LIN {X 0,Y 573.208,Z 412.078,A -85,B 0,C 180,E1 -2311.434,E2 -2311.434} C_VEL
LIN {X 0,Y 573.228,Z 412.081,A -85,B 0,C 180,E1 -2314.589,E2 -2314.589} C_VEL
LIN {X 0,Y 573.218,Z 412.079,A -85,B 0,C 180,E1 -2317.661,E2 -2317.661} C_VEL
LIN {X 0,Y 573.204,Z 412.085,A -85,B 0,C 180,E1 -2319.921,E2 -2319.921} C_VEL
LIN {X 0,Y 573.193,Z 412.081,A -85,B 0,C 180,E1 -2323.014,E2 -2323.014} C_VEL
LIN {X 0,Y 573.247,Z 412.08,A -85,B 0,C 180,E1 -2325.806,E2 -2325.806} C_VEL
LIN {X 0,Y 573.224,Z 412.077,A -85,B 0,C 180,E1 -2328.768,E2 -2328.768} C_VEL
LIN {X 0,Y 573.234,Z 412.08,A -85,B 0,C 180,E1 -2331.54,E2 -2331.54} C_VEL
LIN {X 0,Y 573.262,Z 412.075,A -85,B 0,C 180,E1 -2334.371,E2 -2334.371} C_VEL
LIN {X 0,Y 573.309,Z 412.075,A -85,B 0,C 180,E1 -2337.892,E2 -2337.892} C_VEL
LIN {X 0,Y 573.268,Z 412.217,A -85,B 0,C 180,E1 -2339.122,E2 -2339.122} C_VEL
LIN {X 0,Y 573.209,Z 422.347,A -85,B 0,C 180,E1 -2341.229,E2 -2341.229} C_VEL
LIN {X 0,Y 574.074,Z 428.345,A -85,B 0,C 180,E1 -2341.337,E2 -2341.337} C_VEL
LIN {X 0,Y 573.848,Z 528.439,A -85,B 0,C 180,E1 -2342.61,E2 -2342.61} C_VEL
LIN {X 0,Y 573.75,Z 541.247,A -85,B 0,C 180,E1 -2342.918,E2 -2342.918} C_VEL
LIN {X 0,Y 573.682,Z 553.267,A -85,B 0,C 180,E1 -2343.336,E2 -2343.336} C_VEL
LIN {X 0,Y 573.54,Z 566.249,A -85,B 0,C 180,E1 -2343.952,E2 -2343.952} C_VEL
LIN {X 0,Y 573.376,Z 577.571,A -85,B 0,C 180,E1 -2344.658,E2 -2344.658} C_VEL
LIN {X 0,Y 573.327,Z 586.745,A -85,B 0,C 180,E1 -2345.363,E2 -2345.363} C_VEL
LIN {X 0,Y 573.226,Z 595.361,A -85,B 0,C 180,E1 -2346.158,E2 -2346.158} C_VEL
LIN {X 0,Y 573.165,Z 603.328,A -85,B 0,C 180,E1 -2347.043,E2 -2347.043} C_VEL
LIN {X 0,Y 573.122,Z 611.174,A -85,B 0,C 180,E1 -2348.107,E2 -2348.107} C_VEL
LIN {X 0,Y 573.018,Z 617.448,A -85,B 0,C 180,E1 -2349.175,E2 -2349.175} C_VEL
LIN {X 0,Y 573.002,Z 622.437,A -85,B 0,C 180,E1 -2350.244,E2 -2350.244} C_VEL
LIN {X 0,Y 572.984,Z 626.292,A -85,B 0,C 180,E1 -2351.318,E2 -2351.318} C_VEL
LIN {X 0,Y 572.952,Z 628.329,A -85,B 0,C 180,E1 -2352.036,E2 -2352.036} C_VEL
LIN {X 0,Y 572.946,Z 629.872,A -85,B 0,C 180,E1 -2352.756,E2 -2352.756} C_VEL
LIN {X 0,Y 572.981,Z 631.694,A -85,B 0,C 180,E1 -2354.2,E2 -2354.2} C_VEL
LIN {X 0,Y 572.906,Z 631.98,A -85,B 0,C 180,E1 -2354.928,E2 -2354.928} C_VEL
LIN {X 0,Y 572.917,Z 631.812,A -85,B 0,C 180,E1 -2355.657,E2 -2355.657} C_VEL
LIN {X 0,Y 572.942,Z 630.599,A -85,B 0,C 180,E1 -2356.904,E2 -2356.904} C_VEL
LIN {X 0,Y 572.952,Z 628.779,A -85,B 0,C 180,E1 -2357.858,E2 -2357.858} C_VEL
LIN {X 0,Y 572.974,Z 624.979,A -85,B 0,C 180,E1 -2359.183,E2 -2359.183} C_VEL
LIN {X 0,Y 573.014,Z 619.717,A -85,B 0,C 180,E1 -2360.46,E2 -2360.46} C_VEL
LIN {X 0,Y 573.092,Z 613.633,A -85,B 0,C 180,E1 -2361.586,E2 -2361.586} C_VEL
LIN {X 0,Y 573.121,Z 605.915,A -85,B 0,C 180,E1 -2362.723,E2 -2362.723} C_VEL
LIN {X 0,Y 573.121,Z 605.356,A -85,B 0,C 180,E1 -2362.795,E2 -2362.795} C_VEL
LIN {X 0,Y 572.463,Z 601.704,A -85,B 0,C 180,E1 -2363.256,E2 -2363.256} C_VEL
LIN {X 0,Y 569.645,Z 595.469,A -85,B 0,C 180,E1 -2363.977,E2 -2363.977} C_VEL
LIN {X 0,Y 566.893,Z 588.846,A -85,B 0,C 180,E1 -2364.659,E2 -2364.659} C_VEL
LIN {X 0,Y 566.352,Z 584.328,A -85,B 0,C 180,E1 -2365.053,E2 -2365.053} C_VEL
LIN {X 0,Y 566.483,Z 572.018,A -85,B 0,C 180,E1 -2365.933,E2 -2365.933} C_VEL
LIN {X 0,Y 566.64,Z 561.548,A -85,B 0,C 180,E1 -2366.52,E2 -2366.52} C_VEL
LIN {X 0,Y 566.736,Z 550.579,A -85,B 0,C 180,E1 -2367.005,E2 -2367.005} C_VEL
LIN {X 0,Y 566.849,Z 538.8,A -85,B 0,C 180,E1 -2367.393,E2 -2367.393} C_VEL
LIN {X 0,Y 566.936,Z 525.781,A -85,B 0,C 180,E1 -2367.677,E2 -2367.677} C_VEL
LIN {X 0,Y 567.085,Z 427.613,A -85,B 0,C 180,E1 -2368.934,E2 -2368.934} C_VEL
LIN {X 0,Y 566.174,Z 422.329,A -85,B 0,C 180,E1 -2369.039,E2 -2369.039} C_VEL
LIN {X 0,Y 566.194,Z 412.956,A -85,B 0,C 180,E1 -2371.048,E2 -2371.048} C_VEL
LIN {X 0,Y 566.2,Z 412.953,A -85,B 0,C 180,E1 -2373.732,E2 -2373.732} C_VEL
LIN {X 0,Y 566.177,Z 412.961,A -85,B 0,C 180,E1 -2376.572,E2 -2376.572} C_VEL
LIN {X 0,Y 566.212,Z 412.95,A -85,B 0,C 180,E1 -2379.685,E2 -2379.685} C_VEL
LIN {X 0,Y 566.195,Z 412.954,A -85,B 0,C 180,E1 -2382.916,E2 -2382.916} C_VEL
LIN {X 0,Y 566.159,Z 412.96,A -85,B 0,C 180,E1 -2386.053,E2 -2386.053} C_VEL
LIN {X 0,Y 566.16,Z 412.959,A -85,B 0,C 180,E1 -2388.859,E2 -2388.859} C_VEL
LIN {X 0,Y 566.204,Z 412.95,A -85,B 0,C 180,E1 -2391.443,E2 -2391.443} C_VEL
LIN {X 0,Y 566.145,Z 412.966,A -85,B 0,C 180,E1 -2394.306,E2 -2394.306} C_VEL
LIN {X 0,Y 566.213,Z 412.952,A -85,B 0,C 180,E1 -2396.897,E2 -2396.897} C_VEL
LIN {X 0,Y 566.171,Z 412.954,A -85,B 0,C 180,E1 -2399.406,E2 -2399.406} C_VEL
LIN {X 0,Y 566.172,Z 412.956,A -85,B 0,C 180,E1 -2401.855,E2 -2401.855} C_VEL
LIN {X 0,Y 566.196,Z 412.958,A -85,B 0,C 180,E1 -2404.25,E2 -2404.25} C_VEL
LIN {X 0,Y 566.168,Z 412.96,A -85,B 0,C 180,E1 -2406.72,E2 -2406.72} C_VEL
LIN {X 0,Y 566.204,Z 412.951,A -85,B 0,C 180,E1 -2409.662,E2 -2409.662} C_VEL
LIN {X 0,Y 566.178,Z 412.956,A -85,B 0,C 180,E1 -2411.921,E2 -2411.921} C_VEL
LIN {X 0,Y 566.189,Z 412.955,A -85,B 0,C 180,E1 -2414.89,E2 -2414.89} C_VEL
LIN {X 0,Y 566.214,Z 412.95,A -85,B 0,C 180,E1 -2417.818,E2 -2417.818} C_VEL
LIN {X 0,Y 566.174,Z 412.957,A -85,B 0,C 180,E1 -2419.992,E2 -2419.992} C_VEL
LIN {X 0,Y 566.213,Z 412.953,A -85,B 0,C 180,E1 -2422.87,E2 -2422.87} C_VEL
LIN {X 0,Y 566.263,Z 412.945,A -85,B 0,C 180,E1 -2425.016,E2 -2425.016} C_VEL
LIN {X 0,Y 566.281,Z 412.942,A -85,B 0,C 180,E1 -2427.866,E2 -2427.866} C_VEL
LIN {X 0,Y 566.299,Z 412.945,A -85,B 0,C 180,E1 -2430.711,E2 -2430.711} C_VEL
LIN {X 0,Y 566.26,Z 412.948,A -85,B 0,C 180,E1 -2432.845,E2 -2432.845} C_VEL
LIN {X 0,Y 566.247,Z 412.945,A -85,B 0,C 180,E1 -2435.698,E2 -2435.698} C_VEL
LIN {X 0,Y 566.194,Z 412.953,A -85,B 0,C 180,E1 -2437.847,E2 -2437.847} C_VEL
LIN {X 0,Y 566.236,Z 412.953,A -85,B 0,C 180,E1 -2440.73,E2 -2440.73} C_VEL
LIN {X 0,Y 566.189,Z 412.956,A -85,B 0,C 180,E1 -2442.91,E2 -2442.91} C_VEL
LIN {X 0,Y 566.196,Z 412.953,A -85,B 0,C 180,E1 -2445.109,E2 -2445.109} C_VEL
LIN {X 0,Y 566.195,Z 412.952,A -85,B 0,C 180,E1 -2447.332,E2 -2447.332} C_VEL
LIN {X 0,Y 566.207,Z 412.957,A -85,B 0,C 180,E1 -2450.337,E2 -2450.337} C_VEL
LIN {X 0,Y 566.169,Z 412.955,A -85,B 0,C 180,E1 -2453.28,E2 -2453.28} C_VEL
LIN {X 0,Y 566.204,Z 412.95,A -85,B 0,C 180,E1 -2455.749,E2 -2455.749} C_VEL
LIN {X 0,Y 566.184,Z 412.956,A -85,B 0,C 180,E1 -2458.954,E2 -2458.954} C_VEL
LIN {X 0,Y 566.192,Z 412.952,A -85,B 0,C 180,E1 -2461.422,E2 -2461.422} C_VEL
LIN {X 0,Y 566.208,Z 412.951,A -85,B 0,C 180,E1 -2463.956,E2 -2463.956} C_VEL
LIN {X 0,Y 566.182,Z 412.963,A -85,B 0,C 180,E1 -2466.571,E2 -2466.571} C_VEL
LIN {X 0,Y 566.211,Z 412.95,A -85,B 0,C 180,E1 -2469.274,E2 -2469.274} C_VEL
LIN {X 0,Y 566.187,Z 412.955,A -85,B 0,C 180,E1 -2472.09,E2 -2472.09} C_VEL
LIN {X 0,Y 566.167,Z 412.958,A -85,B 0,C 180,E1 -2475.036,E2 -2475.036} C_VEL
LIN {X 0,Y 566.186,Z 412.954,A -85,B 0,C 180,E1 -2477.91,E2 -2477.91} C_VEL
LIN {X 0,Y 566.211,Z 412.957,A -85,B 0,C 180,E1 -2480.726,E2 -2480.726} C_VEL
LIN {X 0,Y 566.181,Z 412.953,A -85,B 0,C 180,E1 -2483.429,E2 -2483.429} C_VEL
LIN {X 0,Y 566.211,Z 412.954,A -85,B 0,C 180,E1 -2486.266,E2 -2486.266} C_VEL
LIN {X 0,Y 566.189,Z 412.957,A -85,B 0,C 180,E1 -2488.924,E2 -2488.924} C_VEL
LIN {X 0,Y 566.191,Z 412.952,A -85,B 0,C 180,E1 -2491.856,E2 -2491.856} C_VEL
LIN {X 0,Y 566.237,Z 412.949,A -85,B 0,C 180,E1 -2495.039,E2 -2495.039} C_VEL
LIN {X 0,Y 566.191,Z 412.955,A -85,B 0,C 180,E1 -2498.137,E2 -2498.137} C_VEL
LIN {X 0,Y 566.23,Z 412.957,A -85,B 0,C 180,E1 -2500.614,E2 -2500.614} C_VEL
LIN {X 0,Y 566.207,Z 412.95,A -85,B 0,C 180,E1 -2503.412,E2 -2503.412} C_VEL
LIN {X 0,Y 566.19,Z 412.958,A -85,B 0,C 180,E1 -2506.359,E2 -2506.359} C_VEL
LIN {X 0,Y 566.235,Z 412.956,A -85,B 0,C 180,E1 -2508.675,E2 -2508.675} C_VEL
LIN {X 0,Y 566.225,Z 412.948,A -85,B 0,C 180,E1 -2511.434,E2 -2511.434} C_VEL
LIN {X 0,Y 566.262,Z 412.947,A -85,B 0,C 180,E1 -2514.302,E2 -2514.302} C_VEL
LIN {X 0,Y 566.282,Z 412.941,A -85,B 0,C 180,E1 -2517.866,E2 -2517.866} C_VEL
LIN {X 0,Y 566.303,Z 412.947,A -85,B 0,C 180,E1 -2520.711,E2 -2520.711} C_VEL
LIN {X 0,Y 566.27,Z 412.949,A -85,B 0,C 180,E1 -2522.846,E2 -2522.846} C_VEL
LIN {X 0,Y 566.251,Z 412.944,A -85,B 0,C 180,E1 -2525.698,E2 -2525.698} C_VEL
LIN {X 0,Y 566.227,Z 412.956,A -85,B 0,C 180,E1 -2528.566,E2 -2528.566} C_VEL
LIN {X 0,Y 566.242,Z 412.946,A -85,B 0,C 180,E1 -2531.454,E2 -2531.454} C_VEL
LIN {X 0,Y 566.235,Z 412.954,A -85,B 0,C 180,E1 -2534.507,E2 -2534.507} C_VEL
LIN {X 0,Y 566.199,Z 412.952,A -85,B 0,C 180,E1 -2537.332,E2 -2537.332} C_VEL
LIN {X 0,Y 566.208,Z 412.954,A -85,B 0,C 180,E1 -2540.337,E2 -2540.337} C_VEL
LIN {X 0,Y 566.17,Z 412.956,A -85,B 0,C 180,E1 -2543.281,E2 -2543.281} C_VEL
LIN {X 0,Y 566.206,Z 412.95,A -85,B 0,C 180,E1 -2545.749,E2 -2545.749} C_VEL
LIN {X 0,Y 566.188,Z 412.958,A -85,B 0,C 180,E1 -2548.954,E2 -2548.954} C_VEL
LIN {X 0,Y 566.193,Z 412.952,A -85,B 0,C 180,E1 -2551.422,E2 -2551.422} C_VEL
LIN {X 0,Y 566.209,Z 412.95,A -85,B 0,C 180,E1 -2553.956,E2 -2553.956} C_VEL
LIN {X 0,Y 566.201,Z 412.958,A -85,B 0,C 180,E1 -2556.57,E2 -2556.57} C_VEL
LIN {X 0,Y 566.214,Z 412.949,A -85,B 0,C 180,E1 -2559.686,E2 -2559.686} C_VEL
LIN {X 0,Y 566.202,Z 412.957,A -85,B 0,C 180,E1 -2562.917,E2 -2562.917} C_VEL
LIN {X 0,Y 566.199,Z 412.952,A -85,B 0,C 180,E1 -2566.049,E2 -2566.049} C_VEL
LIN {X 0,Y 566.205,Z 412.953,A -85,B 0,C 180,E1 -2569.215,E2 -2569.215} C_VEL
LIN {X 0,Y 566.187,Z 412.952,A -85,B 0,C 180,E1 -2571.637,E2 -2571.637} C_VEL
LIN {X 0,Y 566.151,Z 412.96,A -85,B 0,C 180,E1 -2574.307,E2 -2574.307} C_VEL
LIN {X 0,Y 566.221,Z 412.956,A -85,B 0,C 180,E1 -2576.898,E2 -2576.898} C_VEL
LIN {X 0,Y 566.181,Z 412.955,A -85,B 0,C 180,E1 -2579.407,E2 -2579.407} C_VEL
LIN {X 0,Y 566.214,Z 412.951,A -85,B 0,C 180,E1 -2581.858,E2 -2581.858} C_VEL
LIN {X 0,Y 566.221,Z 413.007,A -85,B 0,C 180,E1 -2584.733,E2 -2584.733} C_VEL
LIN {X 0,Y 567.446,Z 419.811,A -85,B 0,C 180,E1 -2585.682,E2 -2585.682} C_VEL
LIN {X 0,Y 567.201,Z 437.42,A -85,B 0,C 180,E1 -2587.987,E2 -2587.987} C_VEL
LIN {X 0,Y 566.912,Z 457.511,A -85,B 0,C 180,E1 -2590.633,E2 -2590.633} C_VEL
LIN {X 0,Y 566.69,Z 477.773,A -85,B 0,C 180,E1 -2593.264,E2 -2593.264} C_VEL
LIN {X 0,Y 566.458,Z 499.265,A -85,B 0,C 180,E1 -2595.988,E2 -2595.988} C_VEL
LIN {X 0,Y 567.166,Z 505.526,A -85,B 0,C 180,E1 -2596.086,E2 -2596.086} C_VEL
LIN {X 0,Y 566.957,Z 607.958,A -85,B 0,C 180,E1 -2597.403,E2 -2597.403} C_VEL
LIN {X 0,Y 566.847,Z 621.226,A -85,B 0,C 180,E1 -2597.719,E2 -2597.719} C_VEL
LIN {X 0,Y 566.719,Z 633.381,A -85,B 0,C 180,E1 -2598.148,E2 -2598.148} C_VEL
LIN {X 0,Y 566.629,Z 645.068,A -85,B 0,C 180,E1 -2598.704,E2 -2598.704} C_VEL
LIN {X 0,Y 566.5,Z 655.912,A -85,B 0,C 180,E1 -2599.366,E2 -2599.366} C_VEL
LIN {X 0,Y 566.335,Z 666.543,A -85,B 0,C 180,E1 -2600.176,E2 -2600.176} C_VEL
LIN {X 0,Y 566.207,Z 676.115,A -85,B 0,C 180,E1 -2601.074,E2 -2601.074} C_VEL
LIN {X 0,Y 566.112,Z 683.962,A -85,B 0,C 180,E1 -2601.972,E2 -2601.972} C_VEL
LIN {X 0,Y 566.003,Z 691.623,A -85,B 0,C 180,E1 -2603.047,E2 -2603.047} C_VEL
LIN {X 0,Y 566.004,Z 698.681,A -85,B 0,C 180,E1 -2604.299,E2 -2604.299} C_VEL
LIN {X 0,Y 565.933,Z 703.373,A -85,B 0,C 180,E1 -2605.37,E2 -2605.37} C_VEL
LIN {X 0,Y 565.927,Z 706.958,A -85,B 0,C 180,E1 -2606.44,E2 -2606.44} C_VEL
LIN {X 0,Y 565.878,Z 708.809,A -85,B 0,C 180,E1 -2607.153,E2 -2607.153} C_VEL
LIN {X 0,Y 565.846,Z 711.186,A -85,B 0,C 180,E1 -2608.577,E2 -2608.577} C_VEL
LIN {X 0,Y 565.839,Z 712,A -85,B 0,C 180,E1 -2610,E2 -2610} C_VEL
LIN {X 0,Y 565.846,Z 711.186,A -85,B 0,C 180,E1 -2611.424,E2 -2611.424} C_VEL
LIN {X 0,Y 565.878,Z 708.809,A -85,B 0,C 180,E1 -2612.848,E2 -2612.848} C_VEL
LIN {X 0,Y 565.926,Z 705.895,A -85,B 0,C 180,E1 -2613.917,E2 -2613.917} C_VEL
LIN {X 0,Y 565.878,Z 701.948,A -85,B 0,C 180,E1 -2614.988,E2 -2614.988} C_VEL
LIN {X 0,Y 566.002,Z 696.865,A -85,B 0,C 180,E1 -2616.059,E2 -2616.059} C_VEL
LIN {X 0,Y 566.04,Z 690.466,A -85,B 0,C 180,E1 -2617.133,E2 -2617.133} C_VEL
LIN {X 0,Y 566.134,Z 682.476,A -85,B 0,C 180,E1 -2618.208,E2 -2618.208} C_VEL
LIN {X 0,Y 566.229,Z 674.333,A -85,B 0,C 180,E1 -2619.106,E2 -2619.106} C_VEL
LIN {X 0,Y 566.345,Z 664.397,A -85,B 0,C 180,E1 -2620.005,E2 -2620.005} C_VEL
LIN {X 0,Y 566.53,Z 653.298,A -85,B 0,C 180,E1 -2620.807,E2 -2620.807} C_VEL
LIN {X 0,Y 566.613,Z 642.17,A -85,B 0,C 180,E1 -2621.447,E2 -2621.447} C_VEL
LIN {X 0,Y 566.722,Z 629.976,A -85,B 0,C 180,E1 -2621.989,E2 -2621.989} C_VEL
LIN {X 0,Y 566.882,Z 617.164,A -85,B 0,C 180,E1 -2622.394,E2 -2622.394} C_VEL
LIN {X 0,Y 566.963,Z 603.581,A -85,B 0,C 180,E1 -2622.665,E2 -2622.665} C_VEL
LIN {X 0,Y 567.027,Z 503.249,A -85,B 0,C 180,E1 -2623.947,E2 -2623.947} C_VEL
LIN {X 0,Y 566.442,Z 498.943,A -85,B 0,C 180,E1 -2624.024,E2 -2624.024} C_VEL
LIN {X 0,Y 566.708,Z 476.505,A -85,B 0,C 180,E1 -2626.9,E2 -2626.9} C_VEL
LIN {X 0,Y 566.959,Z 454.781,A -85,B 0,C 180,E1 -2629.724,E2 -2629.724} C_VEL
LIN {X 0,Y 567.29,Z 434.546,A -85,B 0,C 180,E1 -2632.393,E2 -2632.393} C_VEL
LIN {X 0,Y 567.403,Z 419.645,A -85,B 0,C 180,E1 -2634.321,E2 -2634.321} C_VEL
LIN {X 0,Y 566.219,Z 412.959,A -85,B 0,C 180,E1 -2635.263,E2 -2635.263} C_VEL
LIN {X 0,Y 566.207,Z 412.953,A -85,B 0,C 180,E1 -2638.202,E2 -2638.202} C_VEL
LIN {X 0,Y 566.195,Z 412.963,A -85,B 0,C 180,E1 -2641.076,E2 -2641.076} C_VEL
LIN {X 0,Y 566.216,Z 412.952,A -85,B 0,C 180,E1 -2643.734,E2 -2643.734} C_VEL
LIN {X 0,Y 566.203,Z 412.956,A -85,B 0,C 180,E1 -2646.57,E2 -2646.57} C_VEL
LIN {X 0,Y 566.219,Z 412.95,A -85,B 0,C 180,E1 -2649.686,E2 -2649.686} C_VEL
LIN {X 0,Y 566.202,Z 412.959,A -85,B 0,C 180,E1 -2652.917,E2 -2652.917} C_VEL
LIN {X 0,Y 566.198,Z 412.953,A -85,B 0,C 180,E1 -2656.049,E2 -2656.049} C_VEL
LIN {X 0,Y 566.207,Z 412.952,A -85,B 0,C 180,E1 -2659.215,E2 -2659.215} C_VEL
LIN {X 0,Y 566.184,Z 412.953,A -85,B 0,C 180,E1 -2661.637,E2 -2661.637} C_VEL
LIN {X 0,Y 566.147,Z 412.964,A -85,B 0,C 180,E1 -2664.307,E2 -2664.307} C_VEL
LIN {X 0,Y 566.215,Z 412.952,A -85,B 0,C 180,E1 -2666.897,E2 -2666.897} C_VEL
LIN {X 0,Y 566.172,Z 412.955,A -85,B 0,C 180,E1 -2669.407,E2 -2669.407} C_VEL
LIN {X 0,Y 566.174,Z 412.957,A -85,B 0,C 180,E1 -2671.855,E2 -2671.855} C_VEL
LIN {X 0,Y 566.19,Z 412.961,A -85,B 0,C 180,E1 -2674.25,E2 -2674.25} C_VEL
LIN {X 0,Y 566.163,Z 412.956,A -85,B 0,C 180,E1 -2677.368,E2 -2677.368} C_VEL
LIN {X 0,Y 566.154,Z 412.96,A -85,B 0,C 180,E1 -2679.661,E2 -2679.661} C_VEL
LIN {X 0,Y 566.152,Z 412.96,A -85,B 0,C 180,E1 -2682.667,E2 -2682.667} C_VEL
LIN {X 0,Y 566.217,Z 412.953,A -85,B 0,C 180,E1 -2685.626,E2 -2685.626} C_VEL
LIN {X 0,Y 566.19,Z 412.954,A -85,B 0,C 180,E1 -2688.701,E2 -2688.701} C_VEL
LIN {X 0,Y 566.185,Z 412.957,A -85,B 0,C 180,E1 -2691.434,E2 -2691.434} C_VEL
LIN {X 0,Y 566.232,Z 412.952,A -85,B 0,C 180,E1 -2694.301,E2 -2694.301} C_VEL
LIN {X 0,Y 566.28,Z 412.951,A -85,B 0,C 180,E1 -2697.866,E2 -2697.866} C_VEL
LIN {X 0,Y 566.225,Z 413.125,A -85,B 0,C 180,E1 -2699.111,E2 -2699.111} C_VEL
LIN {X 0,Y 566.196,Z 422.422,A -85,B 0,C 180,E1 -2701.067,E2 -2701.067} C_VEL
LIN {X 0,Y 567.178,Z 429.028,A -85,B 0,C 180,E1 -2701.176,E2 -2701.176} C_VEL
LIN {X 0,Y 566.932,Z 528.869,A -85,B 0,C 180,E1 -2702.464,E2 -2702.464} C_VEL
LIN {X 0,Y 566.791,Z 540.783,A -85,B 0,C 180,E1 -2702.754,E2 -2702.754} C_VEL
LIN {X 0,Y 566.745,Z 552.336,A -85,B 0,C 180,E1 -2703.154,E2 -2703.154} C_VEL
LIN {X 0,Y 566.614,Z 564.791,A -85,B 0,C 180,E1 -2703.734,E2 -2703.734} C_VEL
LIN {X 0,Y 566.42,Z 576.43,A -85,B 0,C 180,E1 -2704.448,E2 -2704.448} C_VEL
LIN {X 0,Y 566.342,Z 585.79,A -85,B 0,C 180,E1 -2705.162,E2 -2705.162} C_VEL
LIN {X 0,Y 566.181,Z 593.677,A -85,B 0,C 180,E1 -2705.878,E2 -2705.878} C_VEL
LIN {X 0,Y 566.14,Z 601.506,A -85,B 0,C 180,E1 -2706.726,E2 -2706.726} C_VEL
LIN {X 0,Y 566.06,Z 608.764,A -85,B 0,C 180,E1 -2707.67,E2 -2707.67} C_VEL
LIN {X 0,Y 565.977,Z 615.551,A -85,B 0,C 180,E1 -2708.749,E2 -2708.749} C_VEL
LIN {X 0,Y 565.94,Z 621.749,A -85,B 0,C 180,E1 -2710.012,E2 -2710.012} C_VEL
LIN {X 0,Y 565.914,Z 625.953,A -85,B 0,C 180,E1 -2711.159,E2 -2711.159} C_VEL
LIN {X 0,Y 565.869,Z 628.757,A -85,B 0,C 180,E1 -2712.189,E2 -2712.189} C_VEL
LIN {X 0,Y 565.845,Z 630.225,A -85,B 0,C 180,E1 -2712.919,E2 -2712.919} C_VEL
LIN {X 0,Y 565.854,Z 631.775,A -85,B 0,C 180,E1 -2714.355,E2 -2714.355} C_VEL
LIN {X 0,Y 565.808,Z 631.99,A -85,B 0,C 180,E1 -2715.12,E2 -2715.12} C_VEL
LIN {X 0,Y 565.812,Z 631.721,A -85,B 0,C 180,E1 -2715.859,E2 -2715.859} C_VEL
LIN {X 0,Y 565.858,Z 630.503,A -85,B 0,C 180,E1 -2716.991,E2 -2716.991} C_VEL
LIN {X 0,Y 565.893,Z 627.34,A -85,B 0,C 180,E1 -2718.463,E2 -2718.463} C_VEL
LIN {X 0,Y 565.889,Z 623.655,A -85,B 0,C 180,E1 -2719.592,E2 -2719.592} C_VEL
LIN {X 0,Y 565.948,Z 618.739,A -85,B 0,C 180,E1 -2720.727,E2 -2720.727} C_VEL
LIN {X 0,Y 566.009,Z 612.427,A -85,B 0,C 180,E1 -2721.87,E2 -2721.87} C_VEL
LIN {X 0,Y 566.074,Z 604.569,A -85,B 0,C 180,E1 -2722.996,E2 -2722.996} C_VEL
LIN {X 0,Y 566.185,Z 595.911,A -85,B 0,C 180,E1 -2723.987,E2 -2723.987} C_VEL
LIN {X 0,Y 566.28,Z 587.734,A -85,B 0,C 180,E1 -2724.763,E2 -2724.763} C_VEL
LIN {X 0,Y 566.352,Z 584.328,A -85,B 0,C 180,E1 -2725.053,E2 -2725.053} C_VEL
LIN {X 0,Y 565.807,Z 579.764,A -85,B 0,C 180,E1 -2725.428,E2 -2725.428} C_VEL
LIN {X 0,Y 563.079,Z 572.097,A -85,B 0,C 180,E1 -2726.003,E2 -2726.003} C_VEL
LIN {X 0,Y 560.399,Z 564.021,A -85,B 0,C 180,E1 -2726.524,E2 -2726.524} C_VEL
LIN {X 0,Y 559.712,Z 558.815,A -85,B 0,C 180,E1 -2726.799,E2 -2726.799} C_VEL
LIN {X 0,Y 559.838,Z 546.217,A -85,B 0,C 180,E1 -2727.322,E2 -2727.322} C_VEL
LIN {X 0,Y 559.97,Z 533.035,A -85,B 0,C 180,E1 -2727.695,E2 -2727.695} C_VEL
LIN {X 0,Y 560.063,Z 518.03,A -85,B 0,C 180,E1 -2727.944,E2 -2727.944} C_VEL
LIN {X 0,Y 560.181,Z 428.464,A -85,B 0,C 180,E1 -2729.098,E2 -2729.098} C_VEL
LIN {X 0,Y 559.125,Z 422.3,A -85,B 0,C 180,E1 -2729.226,E2 -2729.226} C_VEL
LIN {X 0,Y 559.16,Z 413.833,A -85,B 0,C 180,E1 -2731.051,E2 -2731.051} C_VEL
LIN {X 0,Y 559.158,Z 413.832,A -85,B 0,C 180,E1 -2733.947,E2 -2733.947} C_VEL
LIN {X 0,Y 559.127,Z 413.832,A -85,B 0,C 180,E1 -2737.11,E2 -2737.11} C_VEL
LIN {X 0,Y 559.16,Z 413.831,A -85,B 0,C 180,E1 -2739.941,E2 -2739.941} C_VEL
LIN {X 0,Y 559.152,Z 413.833,A -85,B 0,C 180,E1 -2742.744,E2 -2742.744} C_VEL
LIN {X 0,Y 559.126,Z 413.833,A -85,B 0,C 180,E1 -2745.764,E2 -2745.764} C_VEL
LIN {X 0,Y 559.123,Z 413.839,A -85,B 0,C 180,E1 -2748.226,E2 -2748.226} C_VEL
LIN {X 0,Y 559.172,Z 413.827,A -85,B 0,C 180,E1 -2751.192,E2 -2751.192} C_VEL
LIN {X 0,Y 559.118,Z 413.834,A -85,B 0,C 180,E1 -2753.787,E2 -2753.787} C_VEL
LIN {X 0,Y 559.163,Z 413.838,A -85,B 0,C 180,E1 -2756.425,E2 -2756.425} C_VEL
LIN {X 0,Y 559.151,Z 413.831,A -85,B 0,C 180,E1 -2758.98,E2 -2758.98} C_VEL
LIN {X 0,Y 559.119,Z 413.833,A -85,B 0,C 180,E1 -2761.629,E2 -2761.629} C_VEL
LIN {X 0,Y 559.16,Z 413.83,A -85,B 0,C 180,E1 -2763.902,E2 -2763.902} C_VEL
LIN {X 0,Y 559.137,Z 413.839,A -85,B 0,C 180,E1 -2766.573,E2 -2766.573} C_VEL
LIN {X 0,Y 559.175,Z 413.826,A -85,B 0,C 180,E1 -2769.395,E2 -2769.395} C_VEL
LIN {X 0,Y 559.127,Z 413.832,A -85,B 0,C 180,E1 -2771.685,E2 -2771.685} C_VEL
LIN {X 0,Y 559.141,Z 413.833,A -85,B 0,C 180,E1 -2773.947,E2 -2773.947} C_VEL
LIN {X 0,Y 559.158,Z 413.833,A -85,B 0,C 180,E1 -2776.183,E2 -2776.183} C_VEL
LIN {X 0,Y 559.193,Z 413.825,A -85,B 0,C 180,E1 -2779.133,E2 -2779.133} C_VEL
LIN {X 0,Y 559.192,Z 413.827,A -85,B 0,C 180,E1 -2782.053,E2 -2782.053} C_VEL
LIN {X 0,Y 559.239,Z 413.821,A -85,B 0,C 180,E1 -2784.953,E2 -2784.953} C_VEL
LIN {X 0,Y 559.252,Z 413.817,A -85,B 0,C 180,E1 -2787.839,E2 -2787.839} C_VEL
LIN {X 0,Y 559.269,Z 413.82,A -85,B 0,C 180,E1 -2790.72,E2 -2790.72} C_VEL
LIN {X 0,Y 559.226,Z 413.823,A -85,B 0,C 180,E1 -2792.881,E2 -2792.881} C_VEL
LIN {X 0,Y 559.218,Z 413.821,A -85,B 0,C 180,E1 -2795.77,E2 -2795.77} C_VEL
LIN {X 0,Y 559.168,Z 413.834,A -85,B 0,C 180,E1 -2798.674,E2 -2798.674} C_VEL
LIN {X 0,Y 559.206,Z 413.822,A -85,B 0,C 180,E1 -2801.6,E2 -2801.6} C_VEL
LIN {X 0,Y 559.202,Z 413.831,A -85,B 0,C 180,E1 -2804.595,E2 -2804.595} C_VEL
LIN {X 0,Y 559.138,Z 413.83,A -85,B 0,C 180,E1 -2807.557,E2 -2807.557} C_VEL
LIN {X 0,Y 559.167,Z 413.828,A -85,B 0,C 180,E1 -2809.837,E2 -2809.837} C_VEL
LIN {X 0,Y 559.14,Z 413.834,A -85,B 0,C 180,E1 -2812.153,E2 -2812.153} C_VEL
LIN {X 0,Y 559.175,Z 413.826,A -85,B 0,C 180,E1 -2815.298,E2 -2815.298} C_VEL
LIN {X 0,Y 559.127,Z 413.832,A -85,B 0,C 180,E1 -2817.715,E2 -2817.715} C_VEL
LIN {X 0,Y 559.152,Z 413.833,A -85,B 0,C 180,E1 -2820.183,E2 -2820.183} C_VEL
LIN {X 0,Y 559.153,Z 413.836,A -85,B 0,C 180,E1 -2822.715,E2 -2822.715} C_VEL
LIN {X 0,Y 559.122,Z 413.833,A -85,B 0,C 180,E1 -2825.324,E2 -2825.324} C_VEL
LIN {X 0,Y 559.13,Z 413.833,A -85,B 0,C 180,E1 -2828.018,E2 -2828.018} C_VEL
LIN {X 0,Y 559.155,Z 413.834,A -85,B 0,C 180,E1 -2830.812,E2 -2830.812} C_VEL
LIN {X 0,Y 559.111,Z 413.834,A -85,B 0,C 180,E1 -2833.737,E2 -2833.737} C_VEL
LIN {X 0,Y 559.136,Z 413.836,A -85,B 0,C 180,E1 -2836.266,E2 -2836.266} C_VEL
LIN {X 0,Y 559.155,Z 413.83,A -85,B 0,C 180,E1 -2839.187,E2 -2839.187} C_VEL
LIN {X 0,Y 559.129,Z 413.833,A -85,B 0,C 180,E1 -2841.982,E2 -2841.982} C_VEL
LIN {X 0,Y 559.128,Z 413.838,A -85,B 0,C 180,E1 -2844.788,E2 -2844.788} C_VEL
LIN {X 0,Y 559.155,Z 413.829,A -85,B 0,C 180,E1 -2847.365,E2 -2847.365} C_VEL
LIN {X 0,Y 559.147,Z 413.832,A -85,B 0,C 180,E1 -2850.143,E2 -2850.143} C_VEL
LIN {X 0,Y 559.159,Z 413.83,A -85,B 0,C 180,E1 -2853.175,E2 -2853.175} C_VEL
LIN {X 0,Y 559.157,Z 413.828,A -85,B 0,C 180,E1 -2855.495,E2 -2855.495} C_VEL
LIN {X 0,Y 559.171,Z 413.837,A -85,B 0,C 180,E1 -2858.624,E2 -2858.624} C_VEL
LIN {X 0,Y 559.16,Z 413.833,A -85,B 0,C 180,E1 -2860.926,E2 -2860.926} C_VEL
LIN {X 0,Y 559.156,Z 413.829,A -85,B 0,C 180,E1 -2863.948,E2 -2863.948} C_VEL
LIN {X 0,Y 559.163,Z 413.83,A -85,B 0,C 180,E1 -2866.184,E2 -2866.184} C_VEL
LIN {X 0,Y 559.206,Z 413.832,A -85,B 0,C 180,E1 -2868.605,E2 -2868.605} C_VEL
LIN {X 0,Y 559.203,Z 413.824,A -85,B 0,C 180,E1 -2872.054,E2 -2872.054} C_VEL
LIN {X 0,Y 559.247,Z 413.822,A -85,B 0,C 180,E1 -2874.953,E2 -2874.953} C_VEL
LIN {X 0,Y 559.253,Z 413.816,A -85,B 0,C 180,E1 -2877.839,E2 -2877.839} C_VEL
LIN {X 0,Y 559.273,Z 413.823,A -85,B 0,C 180,E1 -2880.72,E2 -2880.72} C_VEL
LIN {X 0,Y 559.236,Z 413.824,A -85,B 0,C 180,E1 -2882.881,E2 -2882.881} C_VEL
LIN {X 0,Y 559.222,Z 413.82,A -85,B 0,C 180,E1 -2885.77,E2 -2885.77} C_VEL
LIN {X 0,Y 559.186,Z 413.835,A -85,B 0,C 180,E1 -2888.674,E2 -2888.674} C_VEL
LIN {X 0,Y 559.206,Z 413.822,A -85,B 0,C 180,E1 -2891.601,E2 -2891.601} C_VEL
LIN {X 0,Y 559.201,Z 413.831,A -85,B 0,C 180,E1 -2894.596,E2 -2894.596} C_VEL
LIN {X 0,Y 559.143,Z 413.83,A -85,B 0,C 180,E1 -2897.558,E2 -2897.558} C_VEL
LIN {X 0,Y 559.166,Z 413.827,A -85,B 0,C 180,E1 -2899.838,E2 -2899.838} C_VEL
LIN {X 0,Y 559.141,Z 413.832,A -85,B 0,C 180,E1 -2902.153,E2 -2902.153} C_VEL
LIN {X 0,Y 559.175,Z 413.827,A -85,B 0,C 180,E1 -2905.298,E2 -2905.298} C_VEL
LIN {X 0,Y 559.168,Z 413.831,A -85,B 0,C 180,E1 -2908.381,E2 -2908.381} C_VEL
LIN {X 0,Y 559.146,Z 413.831,A -85,B 0,C 180,E1 -2911.273,E2 -2911.273} C_VEL
LIN {X 0,Y 559.166,Z 413.827,A -85,B 0,C 180,E1 -2913.949,E2 -2913.949} C_VEL
LIN {X 0,Y 559.141,Z 413.834,A -85,B 0,C 180,E1 -2917.109,E2 -2917.109} C_VEL
LIN {X 0,Y 559.16,Z 413.828,A -85,B 0,C 180,E1 -2919.942,E2 -2919.942} C_VEL
LIN {X 0,Y 559.158,Z 413.838,A -85,B 0,C 180,E1 -2922.744,E2 -2922.744} C_VEL
LIN {X 0,Y 559.152,Z 413.829,A -85,B 0,C 180,E1 -2925.761,E2 -2925.761} C_VEL
LIN {X 0,Y 559.164,Z 413.83,A -85,B 0,C 180,E1 -2928.23,E2 -2928.23} C_VEL
LIN {X 0,Y 559.177,Z 413.829,A -85,B 0,C 180,E1 -2931.192,E2 -2931.192} C_VEL
LIN {X 0,Y 559.123,Z 413.832,A -85,B 0,C 180,E1 -2933.788,E2 -2933.788} C_VEL
LIN {X 0,Y 559.164,Z 413.832,A -85,B 0,C 180,E1 -2936.425,E2 -2936.425} C_VEL
LIN {X 0,Y 559.156,Z 413.835,A -85,B 0,C 180,E1 -2938.981,E2 -2938.981} C_VEL
LIN {X 0,Y 559.147,Z 413.832,A -85,B 0,C 180,E1 -2941.623,E2 -2941.623} C_VEL
LIN {X 0,Y 559.212,Z 413.994,A -85,B 0,C 180,E1 -2944.579,E2 -2944.579} C_VEL
LIN {X 0,Y 560.507,Z 420.864,A -85,B 0,C 180,E1 -2945.558,E2 -2945.558} C_VEL
LIN {X 0,Y 560.272,Z 438.578,A -85,B 0,C 180,E1 -2947.894,E2 -2947.894} C_VEL
LIN {X 0,Y 559.98,Z 459.286,A -85,B 0,C 180,E1 -2950.62,E2 -2950.62} C_VEL
LIN {X 0,Y 559.68,Z 481.906,A -85,B 0,C 180,E1 -2953.589,E2 -2953.589} C_VEL
LIN {X 0,Y 559.501,Z 499.265,A -85,B 0,C 180,E1 -2955.81,E2 -2955.81} C_VEL
LIN {X 0,Y 560.278,Z 506.196,A -85,B 0,C 180,E1 -2955.92,E2 -2955.92} C_VEL
LIN {X 0,Y 560.027,Z 607.958,A -85,B 0,C 180,E1 -2957.245,E2 -2957.245} C_VEL
LIN {X 0,Y 559.904,Z 621.226,A -85,B 0,C 180,E1 -2957.564,E2 -2957.564} C_VEL
LIN {X 0,Y 559.766,Z 633.382,A -85,B 0,C 180,E1 -2957.999,E2 -2957.999} C_VEL
LIN {X 0,Y 559.668,Z 644.813,A -85,B 0,C 180,E1 -2958.547,E2 -2958.547} C_VEL
LIN {X 0,Y 559.516,Z 655.91,A -85,B 0,C 180,E1 -2959.232,E2 -2959.232} C_VEL
LIN {X 0,Y 559.315,Z 666.542,A -85,B 0,C 180,E1 -2960.051,E2 -2960.051} C_VEL
LIN {X 0,Y 559.161,Z 676.115,A -85,B 0,C 180,E1 -2960.961,E2 -2960.961} C_VEL
LIN {X 0,Y 559.05,Z 683.962,A -85,B 0,C 180,E1 -2961.87,E2 -2961.87} C_VEL
LIN {X 0,Y 558.943,Z 691.624,A -85,B 0,C 180,E1 -2962.959,E2 -2962.959} C_VEL
LIN {X 0,Y 558.935,Z 698.681,A -85,B 0,C 180,E1 -2964.227,E2 -2964.227} C_VEL
LIN {X 0,Y 558.826,Z 703.373,A -85,B 0,C 180,E1 -2965.311,E2 -2965.311} C_VEL
LIN {X 0,Y 558.836,Z 706.958,A -85,B 0,C 180,E1 -2966.395,E2 -2966.395} C_VEL
LIN {X 0,Y 558.799,Z 708.808,A -85,B 0,C 180,E1 -2967.117,E2 -2967.117} C_VEL
LIN {X 0,Y 558.745,Z 711.185,A -85,B 0,C 180,E1 -2968.559,E2 -2968.559} C_VEL
LIN {X 0,Y 558.74,Z 712,A -85,B 0,C 180,E1 -2970,E2 -2970} C_VEL
LIN {X 0,Y 558.745,Z 711.185,A -85,B 0,C 180,E1 -2971.442,E2 -2971.442} C_VEL
LIN {X 0,Y 558.799,Z 708.809,A -85,B 0,C 180,E1 -2972.884,E2 -2972.884} C_VEL
LIN {X 0,Y 558.844,Z 705.895,A -85,B 0,C 180,E1 -2973.966,E2 -2973.966} C_VEL
LIN {X 0,Y 558.798,Z 701.948,A -85,B 0,C 180,E1 -2975.051,E2 -2975.051} C_VEL
LIN {X 0,Y 558.921,Z 696.865,A -85,B 0,C 180,E1 -2976.136,E2 -2976.136} C_VEL
LIN {X 0,Y 558.978,Z 690.466,A -85,B 0,C 180,E1 -2977.223,E2 -2977.223} C_VEL
LIN {X 0,Y 559.099,Z 682.475,A -85,B 0,C 180,E1 -2978.312,E2 -2978.312} C_VEL
LIN {X 0,Y 559.185,Z 674.332,A -85,B 0,C 180,E1 -2979.221,E2 -2979.221} C_VEL
LIN {X 0,Y 559.355,Z 664.396,A -85,B 0,C 180,E1 -2980.131,E2 -2980.131} C_VEL
LIN {X 0,Y 559.534,Z 653.4,A -85,B 0,C 180,E1 -2980.937,E2 -2980.937} C_VEL
LIN {X 0,Y 559.672,Z 641.455,A -85,B 0,C 180,E1 -2981.628,E2 -2981.628} C_VEL
LIN {X 0,Y 559.817,Z 628.759,A -85,B 0,C 180,E1 -2982.185,E2 -2982.185} C_VEL
LIN {X 0,Y 559.967,Z 615.334,A -85,B 0,C 180,E1 -2982.596,E2 -2982.596} C_VEL
LIN {X 0,Y 560.072,Z 602.062,A -85,B 0,C 180,E1 -2982.847,E2 -2982.847} C_VEL
LIN {X 0,Y 560.245,Z 504.935,A -85,B 0,C 180,E1 -2984.097,E2 -2984.097} C_VEL
LIN {X 0,Y 559.458,Z 498.943,A -85,B 0,C 180,E1 -2984.203,E2 -2984.203} C_VEL
LIN {X 0,Y 559.735,Z 476.827,A -85,B 0,C 180,E1 -2987.074,E2 -2987.074} C_VEL
LIN {X 0,Y 560.04,Z 456.072,A -85,B 0,C 180,E1 -2989.806,E2 -2989.806} C_VEL
LIN {X 0,Y 560.214,Z 440.013,A -85,B 0,C 180,E1 -2991.907,E2 -2991.907} C_VEL
LIN {X 0,Y 560.501,Z 422.028,A -85,B 0,C 180,E1 -2994.246,E2 -2994.246} C_VEL
LIN {X 0,Y 559.898,Z 417.471,A -85,B 0,C 180,E1 -2994.867,E2 -2994.867} C_VEL
LIN {X 0,Y 559.188,Z 413.834,A -85,B 0,C 180,E1 -2995.398,E2 -2995.398} C_VEL
LIN {X 0,Y 559.172,Z 413.83,A -85,B 0,C 180,E1 -2998.381,E2 -2998.381} C_VEL
LIN {X 0,Y 559.15,Z 413.838,A -85,B 0,C 180,E1 -3001.273,E2 -3001.273} C_VEL
LIN {X 0,Y 559.17,Z 413.829,A -85,B 0,C 180,E1 -3003.949,E2 -3003.949} C_VEL
LIN {X 0,Y 559.145,Z 413.837,A -85,B 0,C 180,E1 -3007.109,E2 -3007.109} C_VEL
LIN {X 0,Y 559.164,Z 413.829,A -85,B 0,C 180,E1 -3009.942,E2 -3009.942} C_VEL
LIN {X 0,Y 559.159,Z 413.838,A -85,B 0,C 180,E1 -3012.744,E2 -3012.744} C_VEL
LIN {X 0,Y 559.153,Z 413.829,A -85,B 0,C 180,E1 -3015.761,E2 -3015.761} C_VEL
LIN {X 0,Y 559.164,Z 413.831,A -85,B 0,C 180,E1 -3018.23,E2 -3018.23} C_VEL
LIN {X 0,Y 559.175,Z 413.828,A -85,B 0,C 180,E1 -3021.192,E2 -3021.192} C_VEL
LIN {X 0,Y 559.122,Z 413.833,A -85,B 0,C 180,E1 -3023.788,E2 -3023.788} C_VEL
LIN {X 0,Y 559.164,Z 413.836,A -85,B 0,C 180,E1 -3026.425,E2 -3026.425} C_VEL
LIN {X 0,Y 559.153,Z 413.831,A -85,B 0,C 180,E1 -3028.98,E2 -3028.98} C_VEL
LIN {X 0,Y 559.119,Z 413.834,A -85,B 0,C 180,E1 -3031.629,E2 -3031.629} C_VEL
LIN {X 0,Y 559.13,Z 413.836,A -85,B 0,C 180,E1 -3034.699,E2 -3034.699} C_VEL
LIN {X 0,Y 559.114,Z 413.835,A -85,B 0,C 180,E1 -3037.066,E2 -3037.066} C_VEL
LIN {X 0,Y 559.114,Z 413.835,A -85,B 0,C 180,E1 -3039.393,E2 -3039.393} C_VEL
LIN {X 0,Y 559.109,Z 413.84,A -85,B 0,C 180,E1 -3042.441,E2 -3042.441} C_VEL
LIN {X 0,Y 559.155,Z 413.831,A -85,B 0,C 180,E1 -3045.441,E2 -3045.441} C_VEL
LIN {X 0,Y 559.146,Z 413.832,A -85,B 0,C 180,E1 -3048.638,E2 -3048.638} C_VEL
LIN {X 0,Y 559.15,Z 413.832,A -85,B 0,C 180,E1 -3051.325,E2 -3051.325} C_VEL
LIN {X 0,Y 559.201,Z 413.829,A -85,B 0,C 180,E1 -3054.229,E2 -3054.229} C_VEL
LIN {X 0,Y 559.25,Z 413.827,A -85,B 0,C 180,E1 -3057.839,E2 -3057.839} C_VEL
LIN {X 0,Y 559.188,Z 413.928,A -85,B 0,C 180,E1 -3059.077,E2 -3059.077} C_VEL
LIN {X 0,Y 559.137,Z 422.362,A -85,B 0,C 180,E1 -3060.878,E2 -3060.878} C_VEL
LIN {X 0,Y 560.283,Z 429.716,A -85,B 0,C 180,E1 -3061.011,E2 -3061.011} C_VEL
LIN {X 0,Y 560.019,Z 528.118,A -85,B 0,C 180,E1 -3062.293,E2 -3062.293} C_VEL
LIN {X 0,Y 559.897,Z 540.264,A -85,B 0,C 180,E1 -3062.585,E2 -3062.585} C_VEL
LIN {X 0,Y 559.786,Z 550.266,A -85,B 0,C 180,E1 -3062.924,E2 -3062.924} C_VEL
LIN {X 0,Y 559.711,Z 559.577,A -85,B 0,C 180,E1 -3063.329,E2 -3063.329} C_VEL
LIN {X 0,Y 559.537,Z 569.557,A -85,B 0,C 180,E1 -3063.871,E2 -3063.871} C_VEL
LIN {X 0,Y 559.362,Z 579.041,A -85,B 0,C 180,E1 -3064.504,E2 -3064.504} C_VEL
LIN {X 0,Y 559.278,Z 587.989,A -85,B 0,C 180,E1 -3065.227,E2 -3065.227} C_VEL
LIN {X 0,Y 559.121,Z 597.303,A -85,B 0,C 180,E1 -3066.133,E2 -3066.133} C_VEL
LIN {X 0,Y 559.025,Z 606.278,A -85,B 0,C 180,E1 -3067.222,E2 -3067.222} C_VEL
LIN {X 0,Y 558.942,Z 613.477,A -85,B 0,C 180,E1 -3068.314,E2 -3068.314} C_VEL
LIN {X 0,Y 558.838,Z 619.301,A -85,B 0,C 180,E1 -3069.409,E2 -3069.409} C_VEL
LIN {X 0,Y 558.829,Z 623.903,A -85,B 0,C 180,E1 -3070.507,E2 -3070.507} C_VEL
LIN {X 0,Y 558.799,Z 627.41,A -85,B 0,C 180,E1 -3071.609,E2 -3071.609} C_VEL
LIN {X 0,Y 558.745,Z 630.521,A -85,B 0,C 180,E1 -3073.086,E2 -3073.086} C_VEL
LIN {X 0,Y 558.762,Z 631.798,A -85,B 0,C 180,E1 -3074.42,E2 -3074.42} C_VEL
LIN {X 0,Y 558.711,Z 631.942,A -85,B 0,C 180,E1 -3075.317,E2 -3075.317} C_VEL
LIN {X 0,Y 558.729,Z 631.596,A -85,B 0,C 180,E1 -3076.065,E2 -3076.065} C_VEL
LIN {X 0,Y 558.767,Z 630.41,A -85,B 0,C 180,E1 -3077.077,E2 -3077.077} C_VEL
LIN {X 0,Y 558.779,Z 627.847,A -85,B 0,C 180,E1 -3078.327,E2 -3078.327} C_VEL
LIN {X 0,Y 558.804,Z 624.628,A -85,B 0,C 180,E1 -3079.392,E2 -3079.392} C_VEL
LIN {X 0,Y 558.844,Z 619.604,A -85,B 0,C 180,E1 -3080.617,E2 -3080.617} C_VEL
LIN {X 0,Y 558.931,Z 615.149,A -85,B 0,C 180,E1 -3081.49,E2 -3081.49} C_VEL
LIN {X 0,Y 558.981,Z 608.51,A -85,B 0,C 180,E1 -3082.549,E2 -3082.549} C_VEL
LIN {X 0,Y 559.095,Z 601.026,A -85,B 0,C 180,E1 -3083.526,E2 -3083.526} C_VEL
LIN {X 0,Y 559.181,Z 593.88,A -85,B 0,C 180,E1 -3084.306,E2 -3084.306} C_VEL
LIN {X 0,Y 559.334,Z 584.742,A -85,B 0,C 180,E1 -3085.143,E2 -3085.143} C_VEL
LIN {X 0,Y 559.457,Z 573.418,A -85,B 0,C 180,E1 -3085.983,E2 -3085.983} C_VEL
LIN {X 0,Y 559.665,Z 562.33,A -85,B 0,C 180,E1 -3086.625,E2 -3086.625} C_VEL
LIN {X 0,Y 559.712,Z 558.815,A -85,B 0,C 180,E1 -3086.799,E2 -3086.799} C_VEL
LIN {X 0,Y 559.144,Z 553.503,A -85,B 0,C 180,E1 -3087.058,E2 -3087.058} C_VEL
LIN {X 0,Y 556.451,Z 544.755,A -85,B 0,C 180,E1 -3087.45,E2 -3087.45} C_VEL
LIN {X 0,Y 553.774,Z 535.764,A -85,B 0,C 180,E1 -3087.776,E2 -3087.776} C_VEL
LIN {X 0,Y 553.102,Z 530.074,A -85,B 0,C 180,E1 -3087.92,E2 -3087.92} C_VEL
LIN {X 0,Y 553.204,Z 505.728,A -85,B 0,C 180,E1 -3088.268,E2 -3088.268} C_VEL
LIN {X 0,Y 553.388,Z 429.806,A -85,B 0,C 180,E1 -3089.257,E2 -3089.257} C_VEL
LIN {X 0,Y 552.05,Z 422.345,A -85,B 0,C 180,E1 -3089.402,E2 -3089.402} C_VEL
LIN {X 0,Y 552.133,Z 414.708,A -85,B 0,C 180,E1 -3091.085,E2 -3091.085} C_VEL
LIN {X 0,Y 552.102,Z 414.715,A -85,B 0,C 180,E1 -3094.165,E2 -3094.165} C_VEL
LIN {X 0,Y 552.098,Z 414.712,A -85,B 0,C 180,E1 -3096.748,E2 -3096.748} C_VEL
LIN {X 0,Y 552.129,Z 414.704,A -85,B 0,C 180,E1 -3099.527,E2 -3099.527} C_VEL
LIN {X 0,Y 552.112,Z 414.716,A -85,B 0,C 180,E1 -3102.427,E2 -3102.427} C_VEL
LIN {X 0,Y 552.077,Z 414.71,A -85,B 0,C 180,E1 -3105.56,E2 -3105.56} C_VEL
LIN {X 0,Y 552.083,Z 414.715,A -85,B 0,C 180,E1 -3108.683,E2 -3108.683} C_VEL
LIN {X 0,Y 552.114,Z 414.705,A -85,B 0,C 180,E1 -3111.41,E2 -3111.41} C_VEL
LIN {X 0,Y 552.068,Z 414.719,A -85,B 0,C 180,E1 -3114.562,E2 -3114.562} C_VEL
LIN {X 0,Y 552.115,Z 414.706,A -85,B 0,C 180,E1 -3117.154,E2 -3117.154} C_VEL
LIN {X 0,Y 552.099,Z 414.71,A -85,B 0,C 180,E1 -3119.953,E2 -3119.953} C_VEL
LIN {X 0,Y 552.095,Z 414.71,A -85,B 0,C 180,E1 -3123.009,E2 -3123.009} C_VEL
LIN {X 0,Y 552.087,Z 414.711,A -85,B 0,C 180,E1 -3125.961,E2 -3125.961} C_VEL
LIN {X 0,Y 552.118,Z 414.706,A -85,B 0,C 180,E1 -3129.119,E2 -3129.119} C_VEL
LIN {X 0,Y 552.087,Z 414.709,A -85,B 0,C 180,E1 -3131.443,E2 -3131.443} C_VEL
LIN {X 0,Y 552.088,Z 414.709,A -85,B 0,C 180,E1 -3133.736,E2 -3133.736} C_VEL
LIN {X 0,Y 552.127,Z 414.707,A -85,B 0,C 180,E1 -3136.004,E2 -3136.004} C_VEL
LIN {X 0,Y 552.162,Z 414.702,A -85,B 0,C 180,E1 -3138.993,E2 -3138.993} C_VEL
LIN {X 0,Y 552.147,Z 414.704,A -85,B 0,C 180,E1 -3141.951,E2 -3141.951} C_VEL
LIN {X 0,Y 552.215,Z 414.696,A -85,B 0,C 180,E1 -3144.889,E2 -3144.889} C_VEL
LIN {X 0,Y 552.223,Z 414.693,A -85,B 0,C 180,E1 -3147.812,E2 -3147.812} C_VEL
LIN {X 0,Y 552.24,Z 414.696,A -85,B 0,C 180,E1 -3150.729,E2 -3150.729} C_VEL
LIN {X 0,Y 552.192,Z 414.699,A -85,B 0,C 180,E1 -3152.918,E2 -3152.918} C_VEL
LIN {X 0,Y 552.191,Z 414.697,A -85,B 0,C 180,E1 -3155.844,E2 -3155.844} C_VEL
LIN {X 0,Y 552.139,Z 414.708,A -85,B 0,C 180,E1 -3158.786,E2 -3158.786} C_VEL
LIN {X 0,Y 552.163,Z 414.7,A -85,B 0,C 180,E1 -3161.75,E2 -3161.75} C_VEL
LIN {X 0,Y 552.137,Z 414.709,A -85,B 0,C 180,E1 -3164.748,E2 -3164.748} C_VEL
LIN {X 0,Y 552.097,Z 414.708,A -85,B 0,C 180,E1 -3167.789,E2 -3167.789} C_VEL
LIN {X 0,Y 552.127,Z 414.707,A -85,B 0,C 180,E1 -3170.101,E2 -3170.101} C_VEL
LIN {X 0,Y 552.091,Z 414.717,A -85,B 0,C 180,E1 -3172.451,E2 -3172.451} C_VEL
LIN {X 0,Y 552.138,Z 414.703,A -85,B 0,C 180,E1 -3175.346,E2 -3175.346} C_VEL
LIN {X 0,Y 552.078,Z 414.713,A -85,B 0,C 180,E1 -3178.1,E2 -3178.1} C_VEL
LIN {X 0,Y 552.101,Z 414.716,A -85,B 0,C 180,E1 -3180.609,E2 -3180.609} C_VEL
LIN {X 0,Y 552.112,Z 414.707,A -85,B 0,C 180,E1 -3183.186,E2 -3183.186} C_VEL
LIN {X 0,Y 552.075,Z 414.711,A -85,B 0,C 180,E1 -3185.844,E2 -3185.844} C_VEL
LIN {X 0,Y 552.116,Z 414.715,A -85,B 0,C 180,E1 -3188.589,E2 -3188.589} C_VEL
LIN {X 0,Y 552.12,Z 414.705,A -85,B 0,C 180,E1 -3191.446,E2 -3191.446} C_VEL
LIN {X 0,Y 552.078,Z 414.72,A -85,B 0,C 180,E1 -3194.53,E2 -3194.53} C_VEL
LIN {X 0,Y 552.109,Z 414.706,A -85,B 0,C 180,E1 -3197.587,E2 -3197.587} C_VEL
LIN {X 0,Y 552.128,Z 414.712,A -85,B 0,C 180,E1 -3200.473,E2 -3200.473} C_VEL
LIN {X 0,Y 552.098,Z 414.708,A -85,B 0,C 180,E1 -3203.318,E2 -3203.318} C_VEL
LIN {X 0,Y 552.125,Z 414.705,A -85,B 0,C 180,E1 -3205.939,E2 -3205.939} C_VEL
LIN {X 0,Y 552.119,Z 414.714,A -85,B 0,C 180,E1 -3208.541,E2 -3208.541} C_VEL
LIN {X 0,Y 552.104,Z 414.707,A -85,B 0,C 180,E1 -3211.442,E2 -3211.442} C_VEL
LIN {X 0,Y 552.123,Z 414.71,A -85,B 0,C 180,E1 -3214.355,E2 -3214.355} C_VEL
LIN {X 0,Y 552.098,Z 414.715,A -85,B 0,C 180,E1 -3216.758,E2 -3216.758} C_VEL
LIN {X 0,Y 552.117,Z 414.708,A -85,B 0,C 180,E1 -3219.12,E2 -3219.12} C_VEL
LIN {X 0,Y 552.118,Z 414.705,A -85,B 0,C 180,E1 -3221.444,E2 -3221.444} C_VEL
LIN {X 0,Y 552.108,Z 414.706,A -85,B 0,C 180,E1 -3223.737,E2 -3223.737} C_VEL
LIN {X 0,Y 552.13,Z 414.705,A -85,B 0,C 180,E1 -3226.004,E2 -3226.004} C_VEL
LIN {X 0,Y 552.161,Z 414.704,A -85,B 0,C 180,E1 -3228.993,E2 -3228.993} C_VEL
LIN {X 0,Y 552.157,Z 414.701,A -85,B 0,C 180,E1 -3231.952,E2 -3231.952} C_VEL
LIN {X 0,Y 552.223,Z 414.698,A -85,B 0,C 180,E1 -3234.889,E2 -3234.889} C_VEL
LIN {X 0,Y 552.224,Z 414.692,A -85,B 0,C 180,E1 -3237.812,E2 -3237.812} C_VEL
LIN {X 0,Y 552.243,Z 414.698,A -85,B 0,C 180,E1 -3240.729,E2 -3240.729} C_VEL
LIN {X 0,Y 552.202,Z 414.7,A -85,B 0,C 180,E1 -3242.918,E2 -3242.918} C_VEL
LIN {X 0,Y 552.193,Z 414.696,A -85,B 0,C 180,E1 -3245.844,E2 -3245.844} C_VEL
LIN {X 0,Y 552.153,Z 414.709,A -85,B 0,C 180,E1 -3248.786,E2 -3248.786} C_VEL
LIN {X 0,Y 552.163,Z 414.699,A -85,B 0,C 180,E1 -3251.751,E2 -3251.751} C_VEL
LIN {X 0,Y 552.137,Z 414.712,A -85,B 0,C 180,E1 -3254.748,E2 -3254.748} C_VEL
LIN {X 0,Y 552.1,Z 414.707,A -85,B 0,C 180,E1 -3257.789,E2 -3257.789} C_VEL
LIN {X 0,Y 552.127,Z 414.705,A -85,B 0,C 180,E1 -3260.101,E2 -3260.101} C_VEL
LIN {X 0,Y 552.092,Z 414.714,A -85,B 0,C 180,E1 -3262.451,E2 -3262.451} C_VEL
LIN {X 0,Y 552.137,Z 414.704,A -85,B 0,C 180,E1 -3265.346,E2 -3265.346} C_VEL
LIN {X 0,Y 552.097,Z 414.709,A -85,B 0,C 180,E1 -3268.099,E2 -3268.099} C_VEL
LIN {X 0,Y 552.102,Z 414.715,A -85,B 0,C 180,E1 -3270.609,E2 -3270.609} C_VEL
LIN {X 0,Y 552.112,Z 414.708,A -85,B 0,C 180,E1 -3273.186,E2 -3273.186} C_VEL
LIN {X 0,Y 552.087,Z 414.709,A -85,B 0,C 180,E1 -3275.844,E2 -3275.844} C_VEL
LIN {X 0,Y 552.117,Z 414.713,A -85,B 0,C 180,E1 -3278.589,E2 -3278.589} C_VEL
LIN {X 0,Y 552.121,Z 414.705,A -85,B 0,C 180,E1 -3281.446,E2 -3281.446} C_VEL
LIN {X 0,Y 552.094,Z 414.715,A -85,B 0,C 180,E1 -3284.532,E2 -3284.532} C_VEL
LIN {X 0,Y 552.13,Z 414.704,A -85,B 0,C 180,E1 -3287.585,E2 -3287.585} C_VEL
LIN {X 0,Y 552.133,Z 414.708,A -85,B 0,C 180,E1 -3290.473,E2 -3290.473} C_VEL
LIN {X 0,Y 552.1,Z 414.709,A -85,B 0,C 180,E1 -3293.318,E2 -3293.318} C_VEL
LIN {X 0,Y 552.127,Z 414.704,A -85,B 0,C 180,E1 -3295.939,E2 -3295.939} C_VEL
LIN {X 0,Y 552.121,Z 414.711,A -85,B 0,C 180,E1 -3298.541,E2 -3298.541} C_VEL
LIN {X 0,Y 552.106,Z 414.71,A -85,B 0,C 180,E1 -3301.442,E2 -3301.442} C_VEL
LIN {X 0,Y 552.138,Z 414.711,A -85,B 0,C 180,E1 -3304.37,E2 -3304.37} C_VEL
LIN {X 0,Y 553.543,Z 421.915,A -85,B 0,C 180,E1 -3305.43,E2 -3305.43} C_VEL
LIN {X 0,Y 553.334,Z 439.238,A -85,B 0,C 180,E1 -3307.746,E2 -3307.746} C_VEL
LIN {X 0,Y 553.017,Z 460.593,A -85,B 0,C 180,E1 -3310.561,E2 -3310.561} C_VEL
LIN {X 0,Y 552.701,Z 483.341,A -85,B 0,C 180,E1 -3313.565,E2 -3313.565} C_VEL
LIN {X 0,Y 552.479,Z 498.947,A -85,B 0,C 180,E1 -3315.614,E2 -3315.614} C_VEL
LIN {X 0,Y 553.398,Z 507.315,A -85,B 0,C 180,E1 -3315.756,E2 -3315.756} C_VEL
LIN {X 0,Y 553.103,Z 607.958,A -85,B 0,C 180,E1 -3317.082,E2 -3317.082} C_VEL
LIN {X 0,Y 552.965,Z 621.225,A -85,B 0,C 180,E1 -3317.406,E2 -3317.406} C_VEL
LIN {X 0,Y 552.812,Z 633.376,A -85,B 0,C 180,E1 -3317.845,E2 -3317.845} C_VEL
LIN {X 0,Y 552.684,Z 645.717,A -85,B 0,C 180,E1 -3318.452,E2 -3318.452} C_VEL
LIN {X 0,Y 552.476,Z 657.2,A -85,B 0,C 180,E1 -3319.186,E2 -3319.186} C_VEL
LIN {X 0,Y 552.301,Z 667.607,A -85,B 0,C 180,E1 -3320.016,E2 -3320.016} C_VEL
LIN {X 0,Y 552.126,Z 676.115,A -85,B 0,C 180,E1 -3320.845,E2 -3320.845} C_VEL
LIN {X 0,Y 552.013,Z 683.962,A -85,B 0,C 180,E1 -3321.765,E2 -3321.765} C_VEL
LIN {X 0,Y 551.889,Z 691.623,A -85,B 0,C 180,E1 -3322.868,E2 -3322.868} C_VEL
LIN {X 0,Y 551.867,Z 698.681,A -85,B 0,C 180,E1 -3324.153,E2 -3324.153} C_VEL
LIN {X 0,Y 551.725,Z 703.374,A -85,B 0,C 180,E1 -3325.251,E2 -3325.251} C_VEL
LIN {X 0,Y 551.75,Z 706.959,A -85,B 0,C 180,E1 -3326.349,E2 -3326.349} C_VEL
LIN {X 0,Y 551.723,Z 708.808,A -85,B 0,C 180,E1 -3327.08,E2 -3327.08} C_VEL
LIN {X 0,Y 551.645,Z 711.184,A -85,B 0,C 180,E1 -3328.54,E2 -3328.54} C_VEL
LIN {X 0,Y 551.64,Z 712,A -85,B 0,C 180,E1 -3330,E2 -3330} C_VEL
LIN {X 0,Y 551.645,Z 711.185,A -85,B 0,C 180,E1 -3331.46,E2 -3331.46} C_VEL
LIN {X 0,Y 551.724,Z 708.809,A -85,B 0,C 180,E1 -3332.921,E2 -3332.921} C_VEL
LIN {X 0,Y 551.764,Z 705.895,A -85,B 0,C 180,E1 -3334.017,E2 -3334.017} C_VEL
LIN {X 0,Y 551.723,Z 701.947,A -85,B 0,C 180,E1 -3335.116,E2 -3335.116} C_VEL
LIN {X 0,Y 551.803,Z 696.188,A -85,B 0,C 180,E1 -3336.342,E2 -3336.342} C_VEL
LIN {X 0,Y 551.927,Z 689.234,A -85,B 0,C 180,E1 -3337.5,E2 -3337.5} C_VEL
LIN {X 0,Y 552.082,Z 680.989,A -85,B 0,C 180,E1 -3338.603,E2 -3338.603} C_VEL
LIN {X 0,Y 552.224,Z 672.536,A -85,B 0,C 180,E1 -3339.524,E2 -3339.524} C_VEL
LIN {X 0,Y 552.424,Z 662.09,A -85,B 0,C 180,E1 -3340.445,E2 -3340.445} C_VEL
LIN {X 0,Y 552.606,Z 651.294,A -85,B 0,C 180,E1 -3341.213,E2 -3341.213} C_VEL
LIN {X 0,Y 552.751,Z 640.401,A -85,B 0,C 180,E1 -3341.831,E2 -3341.831} C_VEL
LIN {X 0,Y 552.876,Z 628.755,A -85,B 0,C 180,E1 -3342.34,E2 -3342.34} C_VEL
LIN {X 0,Y 553.045,Z 615.333,A -85,B 0,C 180,E1 -3342.756,E2 -3342.756} C_VEL
LIN {X 0,Y 553.178,Z 602.062,A -85,B 0,C 180,E1 -3343.01,E2 -3343.01} C_VEL
LIN {X 0,Y 553.297,Z 504.837,A -85,B 0,C 180,E1 -3344.279,E2 -3344.279} C_VEL
LIN {X 0,Y 552.448,Z 498.943,A -85,B 0,C 180,E1 -3344.387,E2 -3344.387} C_VEL
LIN {X 0,Y 552.766,Z 477.525,A -85,B 0,C 180,E1 -3347.204,E2 -3347.204} C_VEL
LIN {X 0,Y 553.045,Z 457.955,A -85,B 0,C 180,E1 -3349.774,E2 -3349.774} C_VEL
LIN {X 0,Y 553.261,Z 439.874,A -85,B 0,C 180,E1 -3352.135,E2 -3352.135} C_VEL
LIN {X 0,Y 553.533,Z 422.902,A -85,B 0,C 180,E1 -3354.371,E2 -3354.371} C_VEL
LIN {X 0,Y 552.156,Z 414.709,A -85,B 0,C 180,E1 -3355.529,E2 -3355.529} C_VEL
LIN {X 0,Y 552.128,Z 414.709,A -85,B 0,C 180,E1 -3358.562,E2 -3358.562} C_VEL
LIN {X 0,Y 552.115,Z 414.712,A -85,B 0,C 180,E1 -3361.476,E2 -3361.476} C_VEL
LIN {X 0,Y 552.137,Z 414.706,A -85,B 0,C 180,E1 -3364.171,E2 -3364.171} C_VEL
LIN {X 0,Y 552.109,Z 414.715,A -85,B 0,C 180,E1 -3366.747,E2 -3366.747} C_VEL
LIN {X 0,Y 552.133,Z 414.706,A -85,B 0,C 180,E1 -3369.527,E2 -3369.527} C_VEL
LIN {X 0,Y 552.133,Z 414.709,A -85,B 0,C 180,E1 -3372.426,E2 -3372.426} C_VEL
LIN {X 0,Y 552.097,Z 414.708,A -85,B 0,C 180,E1 -3375.562,E2 -3375.562} C_VEL
LIN {X 0,Y 552.124,Z 414.714,A -85,B 0,C 180,E1 -3378.679,E2 -3378.679} C_VEL
LIN {X 0,Y 552.118,Z 414.706,A -85,B 0,C 180,E1 -3381.411,E2 -3381.411} C_VEL
LIN {X 0,Y 552.075,Z 414.715,A -85,B 0,C 180,E1 -3384.155,E2 -3384.155} C_VEL
LIN {X 0,Y 552.117,Z 414.71,A -85,B 0,C 180,E1 -3386.814,E2 -3386.814} C_VEL
LIN {X 0,Y 552.096,Z 414.708,A -85,B 0,C 180,E1 -3389.39,E2 -3389.39} C_VEL
LIN {X 0,Y 552.066,Z 414.715,A -85,B 0,C 180,E1 -3391.899,E2 -3391.899} C_VEL
LIN {X 0,Y 552.086,Z 414.714,A -85,B 0,C 180,E1 -3394.666,E2 -3394.666} C_VEL
LIN {X 0,Y 552.084,Z 414.711,A -85,B 0,C 180,E1 -3397.549,E2 -3397.549} C_VEL
LIN {X 0,Y 552.086,Z 414.712,A -85,B 0,C 180,E1 -3400.672,E2 -3400.672} C_VEL
LIN {X 0,Y 552.065,Z 414.717,A -85,B 0,C 180,E1 -3403.736,E2 -3403.736} C_VEL
LIN {X 0,Y 552.105,Z 414.716,A -85,B 0,C 180,E1 -3406.004,E2 -3406.004} C_VEL
LIN {X 0,Y 552.122,Z 414.706,A -85,B 0,C 180,E1 -3408.992,E2 -3408.992} C_VEL
LIN {X 0,Y 552.11,Z 414.716,A -85,B 0,C 180,E1 -3411.951,E2 -3411.951} C_VEL
LIN {X 0,Y 552.205,Z 414.697,A -85,B 0,C 180,E1 -3414.889,E2 -3414.889} C_VEL
LIN {X 0,Y 552.221,Z 414.703,A -85,B 0,C 180,E1 -3417.812,E2 -3417.812} C_VEL
LIN {X 0,Y 552.153,Z 414.755,A -85,B 0,C 180,E1 -3419.043,E2 -3419.043} C_VEL
LIN {X 0,Y 552.076,Z 422.321,A -85,B 0,C 180,E1 -3420.684,E2 -3420.684} C_VEL
LIN {X 0,Y 553.406,Z 430.378,A -85,B 0,C 180,E1 -3420.841,E2 -3420.841} C_VEL
LIN {X 0,Y 553.107,Z 528.596,A -85,B 0,C 180,E1 -3422.139,E2 -3422.139} C_VEL
LIN {X 0,Y 552.957,Z 540.541,A -85,B 0,C 180,E1 -3422.436,E2 -3422.436} C_VEL
LIN {X 0,Y 552.828,Z 550.478,A -85,B 0,C 180,E1 -3422.778,E2 -3422.778} C_VEL
LIN {X 0,Y 552.734,Z 559.749,A -85,B 0,C 180,E1 -3423.189,E2 -3423.189} C_VEL
LIN {X 0,Y 552.555,Z 569.694,A -85,B 0,C 180,E1 -3423.737,E2 -3423.737} C_VEL
LIN {X 0,Y 552.385,Z 577.913,A -85,B 0,C 180,E1 -3424.287,E2 -3424.287} C_VEL
LIN {X 0,Y 552.278,Z 585.999,A -85,B 0,C 180,E1 -3424.928,E2 -3424.928} C_VEL
LIN {X 0,Y 552.119,Z 593.845,A -85,B 0,C 180,E1 -3425.661,E2 -3425.661} C_VEL
LIN {X 0,Y 552.022,Z 602.042,A -85,B 0,C 180,E1 -3426.58,E2 -3426.58} C_VEL
LIN {X 0,Y 551.935,Z 608.878,A -85,B 0,C 180,E1 -3427.499,E2 -3427.499} C_VEL
LIN {X 0,Y 551.834,Z 615.653,A -85,B 0,C 180,E1 -3428.606,E2 -3428.606} C_VEL
LIN {X 0,Y 551.759,Z 621.817,A -85,B 0,C 180,E1 -3429.902,E2 -3429.902} C_VEL
LIN {X 0,Y 551.739,Z 625.817,A -85,B 0,C 180,E1 -3431.015,E2 -3431.015} C_VEL
LIN {X 0,Y 551.689,Z 627.95,A -85,B 0,C 180,E1 -3431.761,E2 -3431.761} C_VEL
LIN {X 0,Y 551.658,Z 630.756,A -85,B 0,C 180,E1 -3433.257,E2 -3433.257} C_VEL
LIN {X 0,Y 551.652,Z 631.817,A -85,B 0,C 180,E1 -3434.479,E2 -3434.479} C_VEL
LIN {X 0,Y 551.607,Z 631.854,A -85,B 0,C 180,E1 -3435.519,E2 -3435.519} C_VEL
LIN {X 0,Y 551.634,Z 631.418,A -85,B 0,C 180,E1 -3436.277,E2 -3436.277} C_VEL
LIN {X 0,Y 551.684,Z 630.314,A -85,B 0,C 180,E1 -3437.168,E2 -3437.168} C_VEL
LIN {X 0,Y 551.691,Z 627.272,A -85,B 0,C 180,E1 -3438.571,E2 -3438.571} C_VEL
LIN {X 0,Y 551.732,Z 623.419,A -85,B 0,C 180,E1 -3439.767,E2 -3439.767} C_VEL
LIN {X 0,Y 551.804,Z 618.629,A -85,B 0,C 180,E1 -3440.893,E2 -3440.893} C_VEL
LIN {X 0,Y 551.878,Z 612.295,A -85,B 0,C 180,E1 -3442.066,E2 -3442.066} C_VEL
LIN {X 0,Y 551.966,Z 604.19,A -85,B 0,C 180,E1 -3443.248,E2 -3443.248} C_VEL
LIN {X 0,Y 552.111,Z 595.689,A -85,B 0,C 180,E1 -3444.238,E2 -3444.238} C_VEL
LIN {X 0,Y 552.258,Z 587.904,A -85,B 0,C 180,E1 -3444.996,E2 -3444.996} C_VEL
LIN {X 0,Y 552.378,Z 578.864,A -85,B 0,C 180,E1 -3445.733,E2 -3445.733} C_VEL
LIN {X 0,Y 552.55,Z 570.016,A -85,B 0,C 180,E1 -3446.333,E2 -3446.333} C_VEL
LIN {X 0,Y 552.701,Z 561.202,A -85,B 0,C 180,E1 -3446.829,E2 -3446.829} C_VEL
LIN {X 0,Y 552.851,Z 551.114,A -85,B 0,C 180,E1 -3447.286,E2 -3447.286} C_VEL
LIN {X 0,Y 552.977,Z 541.051,A -85,B 0,C 180,E1 -3447.639,E2 -3447.639} C_VEL
LIN {X 0,Y 553.102,Z 530.074,A -85,B 0,C 180,E1 -3447.92,E2 -3447.92} C_VEL
LIN {X 0,Y 552.464,Z 524.322,A -85,B 0,C 180,E1 -3448.046,E2 -3448.046} C_VEL
LIN {X 0,Y 546.974,Z 505.621,A -85,B 0,C 180,E1 -3448.427,E2 -3448.427} C_VEL
LIN {X 0,Y 546.349,Z 499.807,A -85,B 0,C 180,E1 -3448.515,E2 -3448.515} C_VEL
LIN {X 0,Y 546.404,Z 430.008,A -85,B 0,C 180,E1 -3449.439,E2 -3449.439} C_VEL
LIN {X 0,Y 545.051,Z 422.506,A -85,B 0,C 180,E1 -3449.594,E2 -3449.594} C_VEL
LIN {X 0,Y 545.106,Z 415.584,A -85,B 0,C 180,E1 -3451.198,E2 -3451.198} C_VEL
LIN {X 0,Y 545.06,Z 415.586,A -85,B 0,C 180,E1 -3453.672,E2 -3453.672} C_VEL
LIN {X 0,Y 545.039,Z 415.589,A -85,B 0,C 180,E1 -3456.921,E2 -3456.921} C_VEL
LIN {X 0,Y 545.074,Z 415.582,A -85,B 0,C 180,E1 -3459.319,E2 -3459.319} C_VEL
LIN {X 0,Y 545.056,Z 415.59,A -85,B 0,C 180,E1 -3462.105,E2 -3462.105} C_VEL
LIN {X 0,Y 545.024,Z 415.592,A -85,B 0,C 180,E1 -3464.828,E2 -3464.828} C_VEL
LIN {X 0,Y 545.041,Z 415.589,A -85,B 0,C 180,E1 -3467.893,E2 -3467.893} C_VEL
LIN {X 0,Y 545.079,Z 415.585,A -85,B 0,C 180,E1 -3470.818,E2 -3470.818} C_VEL
LIN {X 0,Y 545.017,Z 415.59,A -85,B 0,C 180,E1 -3473.617,E2 -3473.617} C_VEL
LIN {X 0,Y 545.066,Z 415.592,A -85,B 0,C 180,E1 -3476.328,E2 -3476.328} C_VEL
LIN {X 0,Y 545.065,Z 415.586,A -85,B 0,C 180,E1 -3478.952,E2 -3478.952} C_VEL
LIN {X 0,Y 545.046,Z 415.586,A -85,B 0,C 180,E1 -3481.504,E2 -3481.504} C_VEL
LIN {X 0,Y 545.05,Z 415.594,A -85,B 0,C 180,E1 -3484.502,E2 -3484.502} C_VEL
LIN {X 0,Y 545.033,Z 415.588,A -85,B 0,C 180,E1 -3487.242,E2 -3487.242} C_VEL
LIN {X 0,Y 545.118,Z 415.586,A -85,B 0,C 180,E1 -3490.414,E2 -3490.414} C_VEL
LIN {X 0,Y 545.039,Z 415.587,A -85,B 0,C 180,E1 -3493.52,E2 -3493.52} C_VEL
LIN {X 0,Y 545.083,Z 415.583,A -85,B 0,C 180,E1 -3495.819,E2 -3495.819} C_VEL
LIN {X 0,Y 545.118,Z 415.581,A -85,B 0,C 180,E1 -3498.849,E2 -3498.849} C_VEL
LIN {X 0,Y 545.095,Z 415.581,A -85,B 0,C 180,E1 -3501.846,E2 -3501.846} C_VEL
LIN {X 0,Y 545.192,Z 415.572,A -85,B 0,C 180,E1 -3504.823,E2 -3504.823} C_VEL
LIN {X 0,Y 545.195,Z 415.568,A -85,B 0,C 180,E1 -3507.783,E2 -3507.783} C_VEL
LIN {X 0,Y 545.21,Z 415.571,A -85,B 0,C 180,E1 -3510.738,E2 -3510.738} C_VEL
LIN {X 0,Y 545.158,Z 415.575,A -85,B 0,C 180,E1 -3512.956,E2 -3512.956} C_VEL
LIN {X 0,Y 545.164,Z 415.573,A -85,B 0,C 180,E1 -3515.919,E2 -3515.919} C_VEL
LIN {X 0,Y 545.099,Z 415.583,A -85,B 0,C 180,E1 -3518.9,E2 -3518.9} C_VEL
LIN {X 0,Y 545.106,Z 415.58,A -85,B 0,C 180,E1 -3521.905,E2 -3521.905} C_VEL
LIN {X 0,Y 545.086,Z 415.584,A -85,B 0,C 180,E1 -3524.943,E2 -3524.943} C_VEL
LIN {X 0,Y 545.069,Z 415.586,A -85,B 0,C 180,E1 -3528.026,E2 -3528.026} C_VEL
LIN {X 0,Y 545.093,Z 415.587,A -85,B 0,C 180,E1 -3530.372,E2 -3530.372} C_VEL
LIN {X 0,Y 545.079,Z 415.582,A -85,B 0,C 180,E1 -3533.559,E2 -3533.559} C_VEL
LIN {X 0,Y 545.073,Z 415.585,A -85,B 0,C 180,E1 -3536.001,E2 -3536.001} C_VEL
LIN {X 0,Y 545.069,Z 415.589,A -85,B 0,C 180,E1 -3538.744,E2 -3538.744} C_VEL
LIN {X 0,Y 545.058,Z 415.585,A -85,B 0,C 180,E1 -3541.679,E2 -3541.679} C_VEL
LIN {X 0,Y 545.061,Z 415.594,A -85,B 0,C 180,E1 -3544.564,E2 -3544.564} C_VEL
LIN {X 0,Y 545.031,Z 415.588,A -85,B 0,C 180,E1 -3547.304,E2 -3547.304} C_VEL
LIN {X 0,Y 545.064,Z 415.587,A -85,B 0,C 180,E1 -3550.143,E2 -3550.143} C_VEL
LIN {X 0,Y 545.038,Z 415.595,A -85,B 0,C 180,E1 -3552.694,E2 -3552.694} C_VEL
LIN {X 0,Y 545.031,Z 415.589,A -85,B 0,C 180,E1 -3555.17,E2 -3555.17} C_VEL
LIN {X 0,Y 545.064,Z 415.585,A -85,B 0,C 180,E1 -3557.896,E2 -3557.896} C_VEL
LIN {X 0,Y 545.078,Z 415.588,A -85,B 0,C 180,E1 -3560.818,E2 -3560.818} C_VEL
LIN {X 0,Y 545.033,Z 415.587,A -85,B 0,C 180,E1 -3563.619,E2 -3563.619} C_VEL
LIN {X 0,Y 545.065,Z 415.589,A -85,B 0,C 180,E1 -3566.328,E2 -3566.328} C_VEL
LIN {X 0,Y 545.065,Z 415.588,A -85,B 0,C 180,E1 -3568.952,E2 -3568.952} C_VEL
LIN {X 0,Y 545.082,Z 415.581,A -85,B 0,C 180,E1 -3571.507,E2 -3571.507} C_VEL
LIN {X 0,Y 545.082,Z 415.59,A -85,B 0,C 180,E1 -3574.494,E2 -3574.494} C_VEL
LIN {X 0,Y 545.036,Z 415.588,A -85,B 0,C 180,E1 -3577.242,E2 -3577.242} C_VEL
LIN {X 0,Y 545.116,Z 415.584,A -85,B 0,C 180,E1 -3580.415,E2 -3580.415} C_VEL
LIN {X 0,Y 545.06,Z 415.584,A -85,B 0,C 180,E1 -3583.521,E2 -3583.521} C_VEL
LIN {X 0,Y 545.09,Z 415.581,A -85,B 0,C 180,E1 -3585.82,E2 -3585.82} C_VEL
LIN {X 0,Y 545.117,Z 415.583,A -85,B 0,C 180,E1 -3588.849,E2 -3588.849} C_VEL
LIN {X 0,Y 545.127,Z 415.576,A -85,B 0,C 180,E1 -3591.847,E2 -3591.847} C_VEL
LIN {X 0,Y 545.2,Z 415.574,A -85,B 0,C 180,E1 -3594.823,E2 -3594.823} C_VEL
LIN {X 0,Y 545.195,Z 415.567,A -85,B 0,C 180,E1 -3597.784,E2 -3597.784} C_VEL
LIN {X 0,Y 545.213,Z 415.574,A -85,B 0,C 180,E1 -3600.739,E2 -3600.739} C_VEL
LIN {X 0,Y 545.169,Z 415.576,A -85,B 0,C 180,E1 -3602.956,E2 -3602.956} C_VEL
LIN {X 0,Y 545.166,Z 415.572,A -85,B 0,C 180,E1 -3605.92,E2 -3605.92} C_VEL
LIN {X 0,Y 545.11,Z 415.584,A -85,B 0,C 180,E1 -3608.9,E2 -3608.9} C_VEL
LIN {X 0,Y 545.135,Z 415.575,A -85,B 0,C 180,E1 -3611.904,E2 -3611.904} C_VEL
LIN {X 0,Y 545.086,Z 415.586,A -85,B 0,C 180,E1 -3614.944,E2 -3614.944} C_VEL
LIN {X 0,Y 545.072,Z 415.584,A -85,B 0,C 180,E1 -3618.026,E2 -3618.026} C_VEL
LIN {X 0,Y 545.093,Z 415.585,A -85,B 0,C 180,E1 -3620.372,E2 -3620.372} C_VEL
LIN {X 0,Y 545.079,Z 415.582,A -85,B 0,C 180,E1 -3623.56,E2 -3623.56} C_VEL
LIN {X 0,Y 545.075,Z 415.583,A -85,B 0,C 180,E1 -3626.001,E2 -3626.001} C_VEL
LIN {X 0,Y 545.089,Z 415.59,A -85,B 0,C 180,E1 -3628.748,E2 -3628.748} C_VEL
LIN {X 0,Y 545.058,Z 415.584,A -85,B 0,C 180,E1 -3631.679,E2 -3631.679} C_VEL
LIN {X 0,Y 545.063,Z 415.591,A -85,B 0,C 180,E1 -3634.565,E2 -3634.565} C_VEL
LIN {X 0,Y 545.036,Z 415.589,A -85,B 0,C 180,E1 -3637.304,E2 -3637.304} C_VEL
LIN {X 0,Y 545.065,Z 415.585,A -85,B 0,C 180,E1 -3640.143,E2 -3640.143} C_VEL
LIN {X 0,Y 545.079,Z 415.586,A -85,B 0,C 180,E1 -3643.107,E2 -3643.107} C_VEL
LIN {X 0,Y 545.057,Z 415.587,A -85,B 0,C 180,E1 -3646.226,E2 -3646.226} C_VEL
LIN {X 0,Y 545.083,Z 415.589,A -85,B 0,C 180,E1 -3648.886,E2 -3648.886} C_VEL
LIN {X 0,Y 545.083,Z 415.59,A -85,B 0,C 180,E1 -3650.819,E2 -3650.819} C_VEL
LIN {X 0,Y 545.035,Z 415.587,A -85,B 0,C 180,E1 -3653.619,E2 -3653.619} C_VEL
LIN {X 0,Y 545.067,Z 415.587,A -85,B 0,C 180,E1 -3656.328,E2 -3656.328} C_VEL
LIN {X 0,Y 545.067,Z 415.591,A -85,B 0,C 180,E1 -3658.952,E2 -3658.952} C_VEL
LIN {X 0,Y 545.085,Z 415.584,A -85,B 0,C 180,E1 -3661.507,E2 -3661.507} C_VEL
LIN {X 0,Y 545.107,Z 415.707,A -85,B 0,C 180,E1 -3664.219,E2 -3664.219} C_VEL
LIN {X 0,Y 546.685,Z 424.462,A -85,B 0,C 180,E1 -3665.506,E2 -3665.506} C_VEL
LIN {X 0,Y 546.337,Z 441.809,A -85,B 0,C 180,E1 -3667.85,E2 -3667.85} C_VEL
LIN {X 0,Y 546.029,Z 464.224,A -85,B 0,C 180,E1 -3670.84,E2 -3670.84} C_VEL
LIN {X 0,Y 545.665,Z 487.645,A -85,B 0,C 180,E1 -3673.924,E2 -3673.924} C_VEL
LIN {X 0,Y 545.497,Z 498.994,A -85,B 0,C 180,E1 -3675.432,E2 -3675.432} C_VEL
LIN {X 0,Y 546.535,Z 507.154,A -85,B 0,C 180,E1 -3675.571,E2 -3675.571} C_VEL
LIN {X 0,Y 546.198,Z 607.958,A -85,B 0,C 180,E1 -3676.916,E2 -3676.916} C_VEL
LIN {X 0,Y 546.054,Z 621.225,A -85,B 0,C 180,E1 -3677.244,E2 -3677.244} C_VEL
LIN {X 0,Y 545.857,Z 633.375,A -85,B 0,C 180,E1 -3677.688,E2 -3677.688} C_VEL
LIN {X 0,Y 545.697,Z 645.715,A -85,B 0,C 180,E1 -3678.302,E2 -3678.302} C_VEL
LIN {X 0,Y 545.491,Z 657.198,A -85,B 0,C 180,E1 -3679.045,E2 -3679.045} C_VEL
LIN {X 0,Y 545.289,Z 667.608,A -85,B 0,C 180,E1 -3679.886,E2 -3679.886} C_VEL
LIN {X 0,Y 545.085,Z 676.115,A -85,B 0,C 180,E1 -3680.726,E2 -3680.726} C_VEL
LIN {X 0,Y 544.977,Z 683.962,A -85,B 0,C 180,E1 -3681.658,E2 -3681.658} C_VEL
LIN {X 0,Y 544.823,Z 691.623,A -85,B 0,C 180,E1 -3682.775,E2 -3682.775} C_VEL
LIN {X 0,Y 544.776,Z 698.681,A -85,B 0,C 180,E1 -3684.076,E2 -3684.076} C_VEL
LIN {X 0,Y 544.628,Z 703.374,A -85,B 0,C 180,E1 -3685.189,E2 -3685.189} C_VEL
LIN {X 0,Y 544.669,Z 706.959,A -85,B 0,C 180,E1 -3686.301,E2 -3686.301} C_VEL
LIN {X 0,Y 544.65,Z 708.808,A -85,B 0,C 180,E1 -3687.042,E2 -3687.042} C_VEL
LIN {X 0,Y 544.546,Z 711.183,A -85,B 0,C 180,E1 -3688.521,E2 -3688.521} C_VEL
LIN {X 0,Y 544.541,Z 712,A -85,B 0,C 180,E1 -3690,E2 -3690} C_VEL
LIN {X 0,Y 544.546,Z 711.184,A -85,B 0,C 180,E1 -3691.479,E2 -3691.479} C_VEL
LIN {X 0,Y 544.65,Z 708.809,A -85,B 0,C 180,E1 -3692.959,E2 -3692.959} C_VEL
LIN {X 0,Y 544.684,Z 705.895,A -85,B 0,C 180,E1 -3694.07,E2 -3694.07} C_VEL
LIN {X 0,Y 544.653,Z 701.947,A -85,B 0,C 180,E1 -3695.183,E2 -3695.183} C_VEL
LIN {X 0,Y 544.74,Z 696.703,A -85,B 0,C 180,E1 -3696.328,E2 -3696.328} C_VEL
LIN {X 0,Y 544.837,Z 690.465,A -85,B 0,C 180,E1 -3697.412,E2 -3697.412} C_VEL
LIN {X 0,Y 545.007,Z 682.475,A -85,B 0,C 180,E1 -3698.528,E2 -3698.528} C_VEL
LIN {X 0,Y 545.154,Z 674.331,A -85,B 0,C 180,E1 -3699.461,E2 -3699.461} C_VEL
LIN {X 0,Y 545.369,Z 664.394,A -85,B 0,C 180,E1 -3700.394,E2 -3700.394} C_VEL
LIN {X 0,Y 545.548,Z 654.586,A -85,B 0,C 180,E1 -3701.142,E2 -3701.142} C_VEL
LIN {X 0,Y 545.695,Z 643.573,A -85,B 0,C 180,E1 -3701.817,E2 -3701.817} C_VEL
LIN {X 0,Y 545.897,Z 631.095,A -85,B 0,C 180,E1 -3702.406,E2 -3702.406} C_VEL
LIN {X 0,Y 546.118,Z 618.075,A -85,B 0,C 180,E1 -3702.85,E2 -3702.85} C_VEL
LIN {X 0,Y 546.237,Z 605.083,A -85,B 0,C 180,E1 -3703.131,E2 -3703.131} C_VEL
LIN {X 0,Y 546.503,Z 506.054,A -85,B 0,C 180,E1 -3704.444,E2 -3704.444} C_VEL
LIN {X 0,Y 545.483,Z 498.979,A -85,B 0,C 180,E1 -3704.57,E2 -3704.57} C_VEL
LIN {X 0,Y 545.788,Z 477.588,A -85,B 0,C 180,E1 -3707.388,E2 -3707.388} C_VEL
LIN {X 0,Y 546.073,Z 456.647,A -85,B 0,C 180,E1 -3710.126,E2 -3710.126} C_VEL
LIN {X 0,Y 546.41,Z 435.748,A -85,B 0,C 180,E1 -3712.898,E2 -3712.898} C_VEL
LIN {X 0,Y 546.572,Z 423.778,A -85,B 0,C 180,E1 -3714.5,E2 -3714.5} C_VEL
LIN {X 0,Y 545.103,Z 415.586,A -85,B 0,C 180,E1 -3715.685,E2 -3715.685} C_VEL
LIN {X 0,Y 545.093,Z 415.588,A -85,B 0,C 180,E1 -3718.748,E2 -3718.748} C_VEL
LIN {X 0,Y 545.062,Z 415.589,A -85,B 0,C 180,E1 -3721.679,E2 -3721.679} C_VEL
LIN {X 0,Y 545.076,Z 415.59,A -85,B 0,C 180,E1 -3724.564,E2 -3724.564} C_VEL
LIN {X 0,Y 545.04,Z 415.592,A -85,B 0,C 180,E1 -3727.304,E2 -3727.304} C_VEL
LIN {X 0,Y 545.069,Z 415.586,A -85,B 0,C 180,E1 -3730.143,E2 -3730.143} C_VEL
LIN {X 0,Y 545.082,Z 415.587,A -85,B 0,C 180,E1 -3733.107,E2 -3733.107} C_VEL
LIN {X 0,Y 545.053,Z 415.589,A -85,B 0,C 180,E1 -3736.226,E2 -3736.226} C_VEL
LIN {X 0,Y 545.084,Z 415.588,A -85,B 0,C 180,E1 -3738.885,E2 -3738.885} C_VEL
LIN {X 0,Y 545.082,Z 415.588,A -85,B 0,C 180,E1 -3740.818,E2 -3740.818} C_VEL
LIN {X 0,Y 545.036,Z 415.588,A -85,B 0,C 180,E1 -3743.619,E2 -3743.619} C_VEL
LIN {X 0,Y 545.067,Z 415.591,A -85,B 0,C 180,E1 -3746.328,E2 -3746.328} C_VEL
LIN {X 0,Y 545.066,Z 415.586,A -85,B 0,C 180,E1 -3748.952,E2 -3748.952} C_VEL
LIN {X 0,Y 545.047,Z 415.587,A -85,B 0,C 180,E1 -3751.504,E2 -3751.504} C_VEL
LIN {X 0,Y 545.038,Z 415.594,A -85,B 0,C 180,E1 -3754.505,E2 -3754.505} C_VEL
LIN {X 0,Y 545.03,Z 415.589,A -85,B 0,C 180,E1 -3757.242,E2 -3757.242} C_VEL
LIN {X 0,Y 545.01,Z 415.594,A -85,B 0,C 180,E1 -3759.624,E2 -3759.624} C_VEL
LIN {X 0,Y 545.026,Z 415.591,A -85,B 0,C 180,E1 -3762.748,E2 -3762.748} C_VEL
LIN {X 0,Y 545.065,Z 415.591,A -85,B 0,C 180,E1 -3765.819,E2 -3765.819} C_VEL
LIN {X 0,Y 545.069,Z 415.585,A -85,B 0,C 180,E1 -3768.848,E2 -3768.848} C_VEL
LIN {X 0,Y 545.067,Z 415.593,A -85,B 0,C 180,E1 -3771.846,E2 -3771.846} C_VEL
LIN {X 0,Y 545.163,Z 415.574,A -85,B 0,C 180,E1 -3774.822,E2 -3774.822} C_VEL
LIN {X 0,Y 545.193,Z 415.579,A -85,B 0,C 180,E1 -3777.784,E2 -3777.784} C_VEL
LIN {X 0,Y 545.185,Z 415.739,A -85,B 0,C 180,E1 -3778.938,E2 -3778.938} C_VEL
LIN {X 0,Y 545.08,Z 422.63,A -85,B 0,C 180,E1 -3780.508,E2 -3780.508} C_VEL
LIN {X 0,Y 546.545,Z 431.054,A -85,B 0,C 180,E1 -3780.668,E2 -3780.668} C_VEL
LIN {X 0,Y 546.18,Z 527.779,A -85,B 0,C 180,E1 -3781.959,E2 -3781.959} C_VEL
LIN {X 0,Y 546.046,Z 539.297,A -85,B 0,C 180,E1 -3782.236,E2 -3782.236} C_VEL
LIN {X 0,Y 545.926,Z 549.517,A -85,B 0,C 180,E1 -3782.582,E2 -3782.582} C_VEL
LIN {X 0,Y 545.797,Z 558.094,A -85,B 0,C 180,E1 -3782.952,E2 -3782.952} C_VEL
LIN {X 0,Y 545.617,Z 568.334,A -85,B 0,C 180,E1 -3783.508,E2 -3783.508} C_VEL
LIN {X 0,Y 545.417,Z 576.785,A -85,B 0,C 180,E1 -3784.064,E2 -3784.064} C_VEL
LIN {X 0,Y 545.229,Z 585.069,A -85,B 0,C 180,E1 -3784.713,E2 -3784.713} C_VEL
LIN {X 0,Y 545.167,Z 592.143,A -85,B 0,C 180,E1 -3785.363,E2 -3785.363} C_VEL
LIN {X 0,Y 545.017,Z 600.448,A -85,B 0,C 180,E1 -3786.273,E2 -3786.273} C_VEL
LIN {X 0,Y 544.885,Z 607.538,A -85,B 0,C 180,E1 -3787.206,E2 -3787.206} C_VEL
LIN {X 0,Y 544.816,Z 613.567,A -85,B 0,C 180,E1 -3788.158,E2 -3788.158} C_VEL
LIN {X 0,Y 544.682,Z 619.372,A -85,B 0,C 180,E1 -3789.282,E2 -3789.282} C_VEL
LIN {X 0,Y 544.64,Z 623.96,A -85,B 0,C 180,E1 -3790.408,E2 -3790.408} C_VEL
LIN {X 0,Y 544.659,Z 626.724,A -85,B 0,C 180,E1 -3791.283,E2 -3791.283} C_VEL
LIN {X 0,Y 544.578,Z 628.413,A -85,B 0,C 180,E1 -3791.917,E2 -3791.917} C_VEL
LIN {X 0,Y 544.571,Z 629.931,A -85,B 0,C 180,E1 -3792.673,E2 -3792.673} C_VEL
LIN {X 0,Y 544.588,Z 631.699,A -85,B 0,C 180,E1 -3794.194,E2 -3794.194} C_VEL
LIN {X 0,Y 544.51,Z 631.988,A -85,B 0,C 180,E1 -3794.96,E2 -3794.96} C_VEL
LIN {X 0,Y 544.558,Z 631.18,A -85,B 0,C 180,E1 -3796.495,E2 -3796.495} C_VEL
LIN {X 0,Y 544.581,Z 630.206,A -85,B 0,C 180,E1 -3797.267,E2 -3797.267} C_VEL
LIN {X 0,Y 544.577,Z 628.672,A -85,B 0,C 180,E1 -3798.043,E2 -3798.043} C_VEL
LIN {X 0,Y 544.619,Z 625.57,A -85,B 0,C 180,E1 -3799.212,E2 -3799.212} C_VEL
LIN {X 0,Y 544.685,Z 621.293,A -85,B 0,C 180,E1 -3800.388,E2 -3800.388} C_VEL
LIN {X 0,Y 544.739,Z 616.257,A -85,B 0,C 180,E1 -3801.458,E2 -3801.458} C_VEL
LIN {X 0,Y 544.84,Z 609.708,A -85,B 0,C 180,E1 -3802.566,E2 -3802.566} C_VEL
LIN {X 0,Y 544.963,Z 602.487,A -85,B 0,C 180,E1 -3803.565,E2 -3803.565} C_VEL
LIN {X 0,Y 545.088,Z 595.581,A -85,B 0,C 180,E1 -3804.367,E2 -3804.367} C_VEL
LIN {X 0,Y 545.27,Z 587.358,A -85,B 0,C 180,E1 -3805.172,E2 -3805.172} C_VEL
LIN {X 0,Y 545.374,Z 579.049,A -85,B 0,C 180,E1 -3805.857,E2 -3805.857} C_VEL
LIN {X 0,Y 545.596,Z 569.841,A -85,B 0,C 180,E1 -3806.488,E2 -3806.488} C_VEL
LIN {X 0,Y 545.724,Z 561.792,A -85,B 0,C 180,E1 -3806.95,E2 -3806.95} C_VEL
LIN {X 0,Y 545.913,Z 551.611,A -85,B 0,C 180,E1 -3807.423,E2 -3807.423} C_VEL
LIN {X 0,Y 546.043,Z 541.536,A -85,B 0,C 180,E1 -3807.786,E2 -3807.786} C_VEL
LIN {X 0,Y 546.181,Z 529.865,A -85,B 0,C 180,E1 -3808.091,E2 -3808.091} C_VEL
LIN {X 0,Y 546.311,Z 503.692,A -85,B 0,C 180,E1 -3808.465,E2 -3808.465} C_VEL
LIN {X 0,Y 546.349,Z 499.807,A -85,B 0,C 180,E1 -3808.515,E2 -3808.515} C_VEL
LIN {X 0,Y 545.712,Z 493.998,A -85,B 0,C 180,E1 -3808.608,E2 -3808.608} C_VEL
LIN {X 0,Y 540.129,Z 475.314,A -85,B 0,C 180,E1 -3808.998,E2 -3808.998} C_VEL
LIN {X 0,Y 539.503,Z 469.504,A -85,B 0,C 180,E1 -3809.092,E2 -3809.092} C_VEL
LIN {X 0,Y 539.55,Z 430.943,A -85,B 0,C 180,E1 -3809.612,E2 -3809.612} C_VEL
LIN {X 0,Y 538.082,Z 422.91,A -85,B 0,C 180,E1 -3809.784,E2 -3809.784} C_VEL
LIN {X 0,Y 538.065,Z 416.461,A -85,B 0,C 180,E1 -3811.279,E2 -3811.279} C_VEL
LIN {X 0,Y 538.005,Z 416.471,A -85,B 0,C 180,E1 -3814.174,E2 -3814.174} C_VEL
LIN {X 0,Y 537.988,Z 416.466,A -85,B 0,C 180,E1 -3817.167,E2 -3817.167} C_VEL
LIN {X 0,Y 538.008,Z 416.464,A -85,B 0,C 180,E1 -3819.798,E2 -3819.798} C_VEL
LIN {X 0,Y 537.99,Z 416.469,A -85,B 0,C 180,E1 -3822.789,E2 -3822.789} C_VEL
LIN {X 0,Y 537.996,Z 416.465,A -85,B 0,C 180,E1 -3825.136,E2 -3825.136} C_VEL
LIN {X 0,Y 537.996,Z 416.471,A -85,B 0,C 180,E1 -3828.223,E2 -3828.223} C_VEL
LIN {X 0,Y 538.011,Z 416.463,A -85,B 0,C 180,E1 -3831.169,E2 -3831.169} C_VEL
LIN {X 0,Y 537.967,Z 416.472,A -85,B 0,C 180,E1 -3834.093,E2 -3834.093} C_VEL
LIN {X 0,Y 538.034,Z 416.464,A -85,B 0,C 180,E1 -3836.727,E2 -3836.727} C_VEL
LIN {X 0,Y 538.009,Z 416.463,A -85,B 0,C 180,E1 -3839.56,E2 -3839.56} C_VEL
LIN {X 0,Y 537.998,Z 416.467,A -85,B 0,C 180,E1 -3841.947,E2 -3841.947} C_VEL
LIN {X 0,Y 538.03,Z 416.47,A -85,B 0,C 180,E1 -3844.465,E2 -3844.465} C_VEL
LIN {X 0,Y 538.011,Z 416.465,A -85,B 0,C 180,E1 -3846.928,E2 -3846.928} C_VEL
LIN {X 0,Y 538.083,Z 416.458,A -85,B 0,C 180,E1 -3850.148,E2 -3850.148} C_VEL
LIN {X 0,Y 537.989,Z 416.465,A -85,B 0,C 180,E1 -3853.298,E2 -3853.298} C_VEL
LIN {X 0,Y 538.053,Z 416.457,A -85,B 0,C 180,E1 -3855.63,E2 -3855.63} C_VEL
LIN {X 0,Y 538.079,Z 416.46,A -85,B 0,C 180,E1 -3858.701,E2 -3858.701} C_VEL
LIN {X 0,Y 538.06,Z 416.457,A -85,B 0,C 180,E1 -3861.739,E2 -3861.739} C_VEL
LIN {X 0,Y 538.149,Z 416.45,A -85,B 0,C 180,E1 -3864.755,E2 -3864.755} C_VEL
LIN {X 0,Y 538.167,Z 416.444,A -85,B 0,C 180,E1 -3867.754,E2 -3867.754} C_VEL
LIN {X 0,Y 538.18,Z 416.447,A -85,B 0,C 180,E1 -3870.748,E2 -3870.748} C_VEL
LIN {X 0,Y 538.125,Z 416.451,A -85,B 0,C 180,E1 -3872.994,E2 -3872.994} C_VEL
LIN {X 0,Y 538.119,Z 416.451,A -85,B 0,C 180,E1 -3875.997,E2 -3875.997} C_VEL
LIN {X 0,Y 538.053,Z 416.463,A -85,B 0,C 180,E1 -3878.261,E2 -3878.261} C_VEL
LIN {X 0,Y 538.087,Z 416.453,A -85,B 0,C 180,E1 -3881.598,E2 -3881.598} C_VEL
LIN {X 0,Y 538.061,Z 416.46,A -85,B 0,C 180,E1 -3884.857,E2 -3884.857} C_VEL
LIN {X 0,Y 538.037,Z 416.459,A -85,B 0,C 180,E1 -3887.532,E2 -3887.532} C_VEL
LIN {X 0,Y 538.038,Z 416.467,A -85,B 0,C 180,E1 -3890.651,E2 -3890.651} C_VEL
LIN {X 0,Y 538.002,Z 416.465,A -85,B 0,C 180,E1 -3893.888,E2 -3893.888} C_VEL
LIN {X 0,Y 538.035,Z 416.466,A -85,B 0,C 180,E1 -3896.367,E2 -3896.367} C_VEL
LIN {X 0,Y 538.03,Z 416.464,A -85,B 0,C 180,E1 -3898.933,E2 -3898.933} C_VEL
LIN {X 0,Y 538.01,Z 416.464,A -85,B 0,C 180,E1 -3901.887,E2 -3901.887} C_VEL
LIN {X 0,Y 538.01,Z 416.471,A -85,B 0,C 180,E1 -3904.617,E2 -3904.617} C_VEL
LIN {X 0,Y 537.999,Z 416.465,A -85,B 0,C 180,E1 -3907.169,E2 -3907.169} C_VEL
LIN {X 0,Y 538.01,Z 416.463,A -85,B 0,C 180,E1 -3909.798,E2 -3909.798} C_VEL
LIN {X 0,Y 538.02,Z 416.462,A -85,B 0,C 180,E1 -3911.877,E2 -3911.877} C_VEL
LIN {X 0,Y 538.002,Z 416.465,A -85,B 0,C 180,E1 -3915.137,E2 -3915.137} C_VEL
LIN {X 0,Y 538.023,Z 416.465,A -85,B 0,C 180,E1 -3918.226,E2 -3918.226} C_VEL
LIN {X 0,Y 538.01,Z 416.464,A -85,B 0,C 180,E1 -3921.169,E2 -3921.169} C_VEL
LIN {X 0,Y 537.989,Z 416.468,A -85,B 0,C 180,E1 -3924.089,E2 -3924.089} C_VEL
LIN {X 0,Y 538.03,Z 416.467,A -85,B 0,C 180,E1 -3926.727,E2 -3926.727} C_VEL
LIN {X 0,Y 538.026,Z 416.46,A -85,B 0,C 180,E1 -3929.556,E2 -3929.556} C_VEL
LIN {X 0,Y 538.041,Z 416.468,A -85,B 0,C 180,E1 -3932.651,E2 -3932.651} C_VEL
LIN {X 0,Y 538.023,Z 416.462,A -85,B 0,C 180,E1 -3935.291,E2 -3935.291} C_VEL
LIN {X 0,Y 538.015,Z 416.464,A -85,B 0,C 180,E1 -3938.042,E2 -3938.042} C_VEL
LIN {X 0,Y 538.031,Z 416.464,A -85,B 0,C 180,E1 -3940.94,E2 -3940.94} C_VEL
LIN {X 0,Y 538.009,Z 416.464,A -85,B 0,C 180,E1 -3943.299,E2 -3943.299} C_VEL
LIN {X 0,Y 538.06,Z 416.456,A -85,B 0,C 180,E1 -3945.631,E2 -3945.631} C_VEL
LIN {X 0,Y 538.077,Z 416.463,A -85,B 0,C 180,E1 -3948.702,E2 -3948.702} C_VEL
LIN {X 0,Y 538.083,Z 416.453,A -85,B 0,C 180,E1 -3951.74,E2 -3951.74} C_VEL
LIN {X 0,Y 538.158,Z 416.452,A -85,B 0,C 180,E1 -3954.755,E2 -3954.755} C_VEL
LIN {X 0,Y 538.167,Z 416.443,A -85,B 0,C 180,E1 -3957.755,E2 -3957.755} C_VEL
LIN {X 0,Y 538.183,Z 416.449,A -85,B 0,C 180,E1 -3960.748,E2 -3960.748} C_VEL
LIN {X 0,Y 538.135,Z 416.451,A -85,B 0,C 180,E1 -3962.995,E2 -3962.995} C_VEL
LIN {X 0,Y 538.12,Z 416.45,A -85,B 0,C 180,E1 -3965.997,E2 -3965.997} C_VEL
LIN {X 0,Y 538.06,Z 416.46,A -85,B 0,C 180,E1 -3969.018,E2 -3969.018} C_VEL
LIN {X 0,Y 538.083,Z 416.455,A -85,B 0,C 180,E1 -3972.063,E2 -3972.063} C_VEL
LIN {X 0,Y 538.046,Z 416.461,A -85,B 0,C 180,E1 -3975.144,E2 -3975.144} C_VEL
LIN {X 0,Y 538.026,Z 416.464,A -85,B 0,C 180,E1 -3978.27,E2 -3978.27} C_VEL
LIN {X 0,Y 538.038,Z 416.468,A -85,B 0,C 180,E1 -3980.652,E2 -3980.652} C_VEL
LIN {X 0,Y 538.003,Z 416.464,A -85,B 0,C 180,E1 -3983.889,E2 -3983.889} C_VEL
LIN {X 0,Y 538.036,Z 416.464,A -85,B 0,C 180,E1 -3986.367,E2 -3986.367} C_VEL
LIN {X 0,Y 538.03,Z 416.466,A -85,B 0,C 180,E1 -3988.933,E2 -3988.933} C_VEL
LIN {X 0,Y 538.01,Z 416.463,A -85,B 0,C 180,E1 -3991.887,E2 -3991.887} C_VEL
LIN {X 0,Y 538.013,Z 416.47,A -85,B 0,C 180,E1 -3994.618,E2 -3994.618} C_VEL
LIN {X 0,Y 538.005,Z 416.466,A -85,B 0,C 180,E1 -3997.17,E2 -3997.17} C_VEL
LIN {X 0,Y 538.022,Z 416.461,A -85,B 0,C 180,E1 -3999.797,E2 -3999.797} C_VEL
LIN {X 0,Y 538.02,Z 416.47,A -85,B 0,C 180,E1 -4002.786,E2 -4002.786} C_VEL
LIN {X 0,Y 538.024,Z 416.461,A -85,B 0,C 180,E1 -4005.926,E2 -4005.926} C_VEL
LIN {X 0,Y 538.049,Z 416.46,A -85,B 0,C 180,E1 -4009.224,E2 -4009.224} C_VEL
LIN {X 0,Y 537.991,Z 416.466,A -85,B 0,C 180,E1 -4012.122,E2 -4012.122} C_VEL
LIN {X 0,Y 537.996,Z 416.472,A -85,B 0,C 180,E1 -4014.916,E2 -4014.916} C_VEL
LIN {X 0,Y 538.02,Z 416.461,A -85,B 0,C 180,E1 -4017.618,E2 -4017.618} C_VEL
LIN {X 0,Y 538.016,Z 416.465,A -85,B 0,C 180,E1 -4020.239,E2 -4020.239} C_VEL
LIN {X 0,Y 538.057,Z 416.467,A -85,B 0,C 180,E1 -4022.796,E2 -4022.796} C_VEL
LIN {X 0,Y 538.054,Z 416.564,A -85,B 0,C 180,E1 -4024.032,E2 -4024.032} C_VEL
LIN {X 0,Y 539.767,Z 425.556,A -85,B 0,C 180,E1 -4025.377,E2 -4025.377} C_VEL
LIN {X 0,Y 539.387,Z 443.216,A -85,B 0,C 180,E1 -4027.799,E2 -4027.799} C_VEL
LIN {X 0,Y 539.047,Z 465.279,A -85,B 0,C 180,E1 -4030.78,E2 -4030.78} C_VEL
LIN {X 0,Y 538.625,Z 488.716,A -85,B 0,C 180,E1 -4033.903,E2 -4033.903} C_VEL
LIN {X 0,Y 538.509,Z 499.121,A -85,B 0,C 180,E1 -4035.249,E2 -4035.249} C_VEL
LIN {X 0,Y 539.655,Z 508.071,A -85,B 0,C 180,E1 -4035.399,E2 -4035.399} C_VEL
LIN {X 0,Y 539.296,Z 607.957,A -85,B 0,C 180,E1 -4036.746,E2 -4036.746} C_VEL
LIN {X 0,Y 539.127,Z 621.224,A -85,B 0,C 180,E1 -4037.077,E2 -4037.077} C_VEL
LIN {X 0,Y 538.935,Z 633.374,A -85,B 0,C 180,E1 -4037.527,E2 -4037.527} C_VEL
LIN {X 0,Y 538.746,Z 644.973,A -85,B 0,C 180,E1 -4038.105,E2 -4038.105} C_VEL
LIN {X 0,Y 538.551,Z 655.905,A -85,B 0,C 180,E1 -4038.807,E2 -4038.807} C_VEL
LIN {X 0,Y 538.282,Z 666.539,A -85,B 0,C 180,E1 -4039.658,E2 -4039.658} C_VEL
LIN {X 0,Y 538.068,Z 676.116,A -85,B 0,C 180,E1 -4040.604,E2 -4040.604} C_VEL
LIN {X 0,Y 537.921,Z 683.962,A -85,B 0,C 180,E1 -4041.548,E2 -4041.548} C_VEL
LIN {X 0,Y 537.754,Z 691.623,A -85,B 0,C 180,E1 -4042.679,E2 -4042.679} C_VEL
LIN {X 0,Y 537.693,Z 698.681,A -85,B 0,C 180,E1 -4043.998,E2 -4043.998} C_VEL
LIN {X 0,Y 537.54,Z 703.374,A -85,B 0,C 180,E1 -4045.125,E2 -4045.125} C_VEL
LIN {X 0,Y 537.591,Z 706.959,A -85,B 0,C 180,E1 -4046.252,E2 -4046.252} C_VEL
LIN {X 0,Y 537.551,Z 708.807,A -85,B 0,C 180,E1 -4047.003,E2 -4047.003} C_VEL
LIN {X 0,Y 537.451,Z 711.183,A -85,B 0,C 180,E1 -4048.502,E2 -4048.502} C_VEL
LIN {X 0,Y 537.442,Z 712,A -85,B 0,C 180,E1 -4050,E2 -4050} C_VEL
LIN {X 0,Y 537.451,Z 711.184,A -85,B 0,C 180,E1 -4051.499,E2 -4051.499} C_VEL
LIN {X 0,Y 537.551,Z 708.809,A -85,B 0,C 180,E1 -4052.998,E2 -4052.998} C_VEL
LIN {X 0,Y 537.603,Z 705.894,A -85,B 0,C 180,E1 -4054.123,E2 -4054.123} C_VEL
LIN {X 0,Y 537.587,Z 701.947,A -85,B 0,C 180,E1 -4055.251,E2 -4055.251} C_VEL
LIN {X 0,Y 537.651,Z 697.08,A -85,B 0,C 180,E1 -4056.335,E2 -4056.335} C_VEL
LIN {X 0,Y 537.791,Z 690.465,A -85,B 0,C 180,E1 -4057.509,E2 -4057.509} C_VEL
LIN {X 0,Y 537.973,Z 682.475,A -85,B 0,C 180,E1 -4058.641,E2 -4058.641} C_VEL
LIN {X 0,Y 538.145,Z 674.33,A -85,B 0,C 180,E1 -4059.585,E2 -4059.585} C_VEL
LIN {X 0,Y 538.366,Z 664.393,A -85,B 0,C 180,E1 -4060.531,E2 -4060.531} C_VEL
LIN {X 0,Y 538.583,Z 654.587,A -85,B 0,C 180,E1 -4061.288,E2 -4061.288} C_VEL
LIN {X 0,Y 538.752,Z 643.545,A -85,B 0,C 180,E1 -4061.973,E2 -4061.973} C_VEL
LIN {X 0,Y 538.98,Z 631.093,A -85,B 0,C 180,E1 -4062.568,E2 -4062.568} C_VEL
LIN {X 0,Y 539.183,Z 618.074,A -85,B 0,C 180,E1 -4063.018,E2 -4063.018} C_VEL
LIN {X 0,Y 539.351,Z 605.083,A -85,B 0,C 180,E1 -4063.301,E2 -4063.301} C_VEL
LIN {X 0,Y 539.588,Z 506.452,A -85,B 0,C 180,E1 -4064.623,E2 -4064.623} C_VEL
LIN {X 0,Y 538.469,Z 498.652,A -85,B 0,C 180,E1 -4064.772,E2 -4064.772} C_VEL
LIN {X 0,Y 538.785,Z 476.568,A -85,B 0,C 180,E1 -4067.671,E2 -4067.671} C_VEL
LIN {X 0,Y 539.079,Z 455.472,A -85,B 0,C 180,E1 -4070.471,E2 -4070.471} C_VEL
LIN {X 0,Y 539.506,Z 433.637,A -85,B 0,C 180,E1 -4073.411,E2 -4073.411} C_VEL
LIN {X 0,Y 539.604,Z 424.654,A -85,B 0,C 180,E1 -4074.632,E2 -4074.632} C_VEL
LIN {X 0,Y 538.073,Z 416.461,A -85,B 0,C 180,E1 -4075.839,E2 -4075.839} C_VEL
LIN {X 0,Y 538.035,Z 416.468,A -85,B 0,C 180,E1 -4078.934,E2 -4078.934} C_VEL
LIN {X 0,Y 538.014,Z 416.467,A -85,B 0,C 180,E1 -4081.887,E2 -4081.887} C_VEL
LIN {X 0,Y 538.025,Z 416.469,A -85,B 0,C 180,E1 -4084.619,E2 -4084.619} C_VEL
LIN {X 0,Y 538.008,Z 416.47,A -85,B 0,C 180,E1 -4087.17,E2 -4087.17} C_VEL
LIN {X 0,Y 538.026,Z 416.462,A -85,B 0,C 180,E1 -4089.797,E2 -4089.797} C_VEL
LIN {X 0,Y 538.023,Z 416.47,A -85,B 0,C 180,E1 -4092.786,E2 -4092.786} C_VEL
LIN {X 0,Y 538.023,Z 416.462,A -85,B 0,C 180,E1 -4095.927,E2 -4095.927} C_VEL
LIN {X 0,Y 538.052,Z 416.46,A -85,B 0,C 180,E1 -4099.253,E2 -4099.253} C_VEL
LIN {X 0,Y 537.992,Z 416.468,A -85,B 0,C 180,E1 -4102.122,E2 -4102.122} C_VEL
LIN {X 0,Y 537.996,Z 416.468,A -85,B 0,C 180,E1 -4104.915,E2 -4104.915} C_VEL
LIN {X 0,Y 538.021,Z 416.462,A -85,B 0,C 180,E1 -4107.617,E2 -4107.617} C_VEL
LIN {X 0,Y 538.004,Z 416.47,A -85,B 0,C 180,E1 -4110.238,E2 -4110.238} C_VEL
LIN {X 0,Y 538.005,Z 416.467,A -85,B 0,C 180,E1 -4112.793,E2 -4112.793} C_VEL
LIN {X 0,Y 537.987,Z 416.467,A -85,B 0,C 180,E1 -4115.289,E2 -4115.289} C_VEL
LIN {X 0,Y 538.018,Z 416.469,A -85,B 0,C 180,E1 -4118.043,E2 -4118.043} C_VEL
LIN {X 0,Y 537.961,Z 416.47,A -85,B 0,C 180,E1 -4120.937,E2 -4120.937} C_VEL
LIN {X 0,Y 537.963,Z 416.47,A -85,B 0,C 180,E1 -4123.297,E2 -4123.297} C_VEL
LIN {X 0,Y 538.033,Z 416.465,A -85,B 0,C 180,E1 -4125.63,E2 -4125.63} C_VEL
LIN {X 0,Y 538.022,Z 416.464,A -85,B 0,C 180,E1 -4128.7,E2 -4128.7} C_VEL
LIN {X 0,Y 538.036,Z 416.468,A -85,B 0,C 180,E1 -4131.739,E2 -4131.739} C_VEL
LIN {X 0,Y 538.122,Z 416.452,A -85,B 0,C 180,E1 -4134.755,E2 -4134.755} C_VEL
LIN {X 0,Y 538.164,Z 416.454,A -85,B 0,C 180,E1 -4137.755,E2 -4137.755} C_VEL
LIN {X 0,Y 538.149,Z 416.604,A -85,B 0,C 180,E1 -4138.784,E2 -4138.784} C_VEL
LIN {X 0,Y 538.105,Z 423.308,A -85,B 0,C 180,E1 -4140.327,E2 -4140.327} C_VEL
LIN {X 0,Y 539.695,Z 431.979,A -85,B 0,C 180,E1 -4140.49,E2 -4140.49} C_VEL
LIN {X 0,Y 539.286,Z 529.346,A -85,B 0,C 180,E1 -4141.82,E2 -4141.82} C_VEL
LIN {X 0,Y 539.09,Z 541.205,A -85,B 0,C 180,E1 -4142.125,E2 -4142.125} C_VEL
LIN {X 0,Y 538.953,Z 551.051,A -85,B 0,C 180,E1 -4142.476,E2 -4142.476} C_VEL
LIN {X 0,Y 538.828,Z 560.255,A -85,B 0,C 180,E1 -4142.897,E2 -4142.897} C_VEL
LIN {X 0,Y 538.674,Z 568.628,A -85,B 0,C 180,E1 -4143.366,E2 -4143.366} C_VEL
LIN {X 0,Y 538.439,Z 577.039,A -85,B 0,C 180,E1 -4143.929,E2 -4143.929} C_VEL
LIN {X 0,Y 538.221,Z 586.294,A -85,B 0,C 180,E1 -4144.681,E2 -4144.681} C_VEL
LIN {X 0,Y 538.085,Z 594.029,A -85,B 0,C 180,E1 -4145.434,E2 -4145.434} C_VEL
LIN {X 0,Y 537.957,Z 601.661,A -85,B 0,C 180,E1 -4146.311,E2 -4146.311} C_VEL
LIN {X 0,Y 537.839,Z 607.72,A -85,B 0,C 180,E1 -4147.131,E2 -4147.131} C_VEL
LIN {X 0,Y 537.739,Z 613.614,A -85,B 0,C 180,E1 -4148.077,E2 -4148.077} C_VEL
LIN {X 0,Y 537.641,Z 618.529,A -85,B 0,C 180,E1 -4149.025,E2 -4149.025} C_VEL
LIN {X 0,Y 537.575,Z 623.284,A -85,B 0,C 180,E1 -4150.166,E2 -4150.166} C_VEL
LIN {X 0,Y 537.577,Z 626.986,A -85,B 0,C 180,E1 -4151.328,E2 -4151.328} C_VEL
LIN {X 0,Y 537.476,Z 630.286,A -85,B 0,C 180,E1 -4152.844,E2 -4152.844} C_VEL
LIN {X 0,Y 537.486,Z 631.771,A -85,B 0,C 180,E1 -4154.385,E2 -4154.385} C_VEL
LIN {X 0,Y 537.419,Z 631.981,A -85,B 0,C 180,E1 -4155.162,E2 -4155.162} C_VEL
LIN {X 0,Y 537.43,Z 631.677,A -85,B 0,C 180,E1 -4155.939,E2 -4155.939} C_VEL
LIN {X 0,Y 537.493,Z 629.816,A -85,B 0,C 180,E1 -4157.502,E2 -4157.502} C_VEL
LIN {X 0,Y 537.515,Z 627.205,A -85,B 0,C 180,E1 -4158.683,E2 -4158.683} C_VEL
LIN {X 0,Y 537.548,Z 624.037,A -85,B 0,C 180,E1 -4159.721,E2 -4159.721} C_VEL
LIN {X 0,Y 537.618,Z 620.362,A -85,B 0,C 180,E1 -4160.668,E2 -4160.668} C_VEL
LIN {X 0,Y 537.678,Z 615.546,A -85,B 0,C 180,E1 -4161.67,E2 -4161.67} C_VEL
LIN {X 0,Y 537.762,Z 609.624,A -85,B 0,C 180,E1 -4162.677,E2 -4162.677} C_VEL
LIN {X 0,Y 537.917,Z 602.494,A -85,B 0,C 180,E1 -4163.675,E2 -4163.675} C_VEL
LIN {X 0,Y 538.053,Z 595.471,A -85,B 0,C 180,E1 -4164.501,E2 -4164.501} C_VEL
LIN {X 0,Y 538.217,Z 588.413,A -85,B 0,C 180,E1 -4165.215,E2 -4165.215} C_VEL
LIN {X 0,Y 538.367,Z 580.418,A -85,B 0,C 180,E1 -4165.902,E2 -4165.902} C_VEL
LIN {X 0,Y 538.576,Z 571.413,A -85,B 0,C 180,E1 -4166.547,E2 -4166.547} C_VEL
LIN {X 0,Y 538.798,Z 561.81,A -85,B 0,C 180,E1 -4167.111,E2 -4167.111} C_VEL
LIN {X 0,Y 538.971,Z 552.873,A -85,B 0,C 180,E1 -4167.538,E2 -4167.538} C_VEL
LIN {X 0,Y 539.117,Z 542.276,A -85,B 0,C 180,E1 -4167.931,E2 -4167.931} C_VEL
LIN {X 0,Y 539.264,Z 530.526,A -85,B 0,C 180,E1 -4168.245,E2 -4168.245} C_VEL
LIN {X 0,Y 539.405,Z 504.767,A -85,B 0,C 180,E1 -4168.622,E2 -4168.622} C_VEL
LIN {X 0,Y 539.503,Z 469.504,A -85,B 0,C 180,E1 -4169.092,E2 -4169.092} C_VEL
LIN {X 0,Y 538.887,Z 463.695,A -85,B 0,C 180,E1 -4169.187,E2 -4169.187} C_VEL
LIN {X 0,Y 533.399,Z 445.005,A -85,B 0,C 180,E1 -4169.591,E2 -4169.591} C_VEL
LIN {X 0,Y 532.786,Z 439.196,A -85,B 0,C 180,E1 -4169.688,E2 -4169.688} C_VEL
LIN {X 0,Y 532.636,Z 431.601,A -85,B 0,C 180,E1 -4169.796,E2 -4169.796} C_VEL
LIN {X 0,Y 531.125,Z 423.363,A -85,B 0,C 180,E1 -4169.967,E2 -4169.967} C_VEL
LIN {X 0,Y 531.013,Z 417.341,A -85,B 0,C 180,E1 -4171.353,E2 -4171.353} C_VEL
LIN {X 0,Y 530.955,Z 417.345,A -85,B 0,C 180,E1 -4173.775,E2 -4173.775} C_VEL
LIN {X 0,Y 530.932,Z 417.351,A -85,B 0,C 180,E1 -4176.56,E2 -4176.56} C_VEL
LIN {X 0,Y 530.97,Z 417.339,A -85,B 0,C 180,E1 -4179.445,E2 -4179.445} C_VEL
LIN {X 0,Y 530.934,Z 417.353,A -85,B 0,C 180,E1 -4182.461,E2 -4182.461} C_VEL
LIN {X 0,Y 530.966,Z 417.34,A -85,B 0,C 180,E1 -4185.45,E2 -4185.45} C_VEL
LIN {X 0,Y 530.961,Z 417.348,A -85,B 0,C 180,E1 -4188.561,E2 -4188.561} C_VEL
LIN {X 0,Y 530.953,Z 417.342,A -85,B 0,C 180,E1 -4191.528,E2 -4191.528} C_VEL
LIN {X 0,Y 530.935,Z 417.353,A -85,B 0,C 180,E1 -4194.378,E2 -4194.378} C_VEL
LIN {X 0,Y 530.969,Z 417.34,A -85,B 0,C 180,E1 -4197.133,E2 -4197.133} C_VEL
LIN {X 0,Y 530.953,Z 417.343,A -85,B 0,C 180,E1 -4199.802,E2 -4199.802} C_VEL
LIN {X 0,Y 530.966,Z 417.349,A -85,B 0,C 180,E1 -4202.478,E2 -4202.478} C_VEL
LIN {X 0,Y 530.958,Z 417.343,A -85,B 0,C 180,E1 -4204.94,E2 -4204.94} C_VEL
LIN {X 0,Y 530.979,Z 417.34,A -85,B 0,C 180,E1 -4207.898,E2 -4207.898} C_VEL
LIN {X 0,Y 530.984,Z 417.344,A -85,B 0,C 180,E1 -4210.677,E2 -4210.677} C_VEL
LIN {X 0,Y 530.956,Z 417.343,A -85,B 0,C 180,E1 -4213.07,E2 -4213.07} C_VEL
LIN {X 0,Y 531.01,Z 417.334,A -85,B 0,C 180,E1 -4215.435,E2 -4215.435} C_VEL
LIN {X 0,Y 531.037,Z 417.339,A -85,B 0,C 180,E1 -4218.549,E2 -4218.549} C_VEL
LIN {X 0,Y 531.035,Z 417.331,A -85,B 0,C 180,E1 -4221.629,E2 -4221.629} C_VEL
LIN {X 0,Y 531.107,Z 417.329,A -85,B 0,C 180,E1 -4224.685,E2 -4224.685} C_VEL
LIN {X 0,Y 531.139,Z 417.319,A -85,B 0,C 180,E1 -4227.725,E2 -4227.725} C_VEL
LIN {X 0,Y 531.151,Z 417.322,A -85,B 0,C 180,E1 -4230.758,E2 -4230.758} C_VEL
LIN {X 0,Y 531.091,Z 417.326,A -85,B 0,C 180,E1 -4233.034,E2 -4233.034} C_VEL
LIN {X 0,Y 531.08,Z 417.329,A -85,B 0,C 180,E1 -4236.077,E2 -4236.077} C_VEL
LIN {X 0,Y 531.014,Z 417.335,A -85,B 0,C 180,E1 -4239.138,E2 -4239.138} C_VEL
LIN {X 0,Y 531.051,Z 417.33,A -85,B 0,C 180,E1 -4241.67,E2 -4241.67} C_VEL
LIN {X 0,Y 531.033,Z 417.335,A -85,B 0,C 180,E1 -4244.955,E2 -4244.955} C_VEL
LIN {X 0,Y 530.982,Z 417.338,A -85,B 0,C 180,E1 -4247.723,E2 -4247.723} C_VEL
LIN {X 0,Y 531.026,Z 417.336,A -85,B 0,C 180,E1 -4250.127,E2 -4250.127} C_VEL
LIN {X 0,Y 530.945,Z 417.352,A -85,B 0,C 180,E1 -4252.573,E2 -4252.573} C_VEL
LIN {X 0,Y 530.989,Z 417.339,A -85,B 0,C 180,E1 -4255.058,E2 -4255.058} C_VEL
LIN {X 0,Y 530.97,Z 417.339,A -85,B 0,C 180,E1 -4257.598,E2 -4257.598} C_VEL
LIN {X 0,Y 530.968,Z 417.344,A -85,B 0,C 180,E1 -4260.197,E2 -4260.197} C_VEL
LIN {X 0,Y 530.967,Z 417.344,A -85,B 0,C 180,E1 -4262.866,E2 -4262.866} C_VEL
LIN {X 0,Y 530.95,Z 417.342,A -85,B 0,C 180,E1 -4265.62,E2 -4265.62} C_VEL
LIN {X 0,Y 530.964,Z 417.348,A -85,B 0,C 180,E1 -4268.653,E2 -4268.653} C_VEL
LIN {X 0,Y 530.989,Z 417.337,A -85,B 0,C 180,E1 -4271.436,E2 -4271.436} C_VEL
LIN {X 0,Y 530.969,Z 417.349,A -85,B 0,C 180,E1 -4274.549,E2 -4274.549} C_VEL
LIN {X 0,Y 530.972,Z 417.34,A -85,B 0,C 180,E1 -4277.835,E2 -4277.835} C_VEL
LIN {X 0,Y 530.984,Z 417.347,A -85,B 0,C 180,E1 -4280.556,E2 -4280.556} C_VEL
LIN {X 0,Y 530.95,Z 417.342,A -85,B 0,C 180,E1 -4283.441,E2 -4283.441} C_VEL
LIN {X 0,Y 530.998,Z 417.344,A -85,B 0,C 180,E1 -4286.494,E2 -4286.494} C_VEL
LIN {X 0,Y 530.974,Z 417.339,A -85,B 0,C 180,E1 -4289.355,E2 -4289.355} C_VEL
LIN {X 0,Y 531.007,Z 417.342,A -85,B 0,C 180,E1 -4292.469,E2 -4292.469} C_VEL
LIN {X 0,Y 530.987,Z 417.342,A -85,B 0,C 180,E1 -4294.942,E2 -4294.942} C_VEL
LIN {X 0,Y 530.971,Z 417.343,A -85,B 0,C 180,E1 -4298.247,E2 -4298.247} C_VEL
LIN {X 0,Y 530.992,Z 417.346,A -85,B 0,C 180,E1 -4300.677,E2 -4300.677} C_VEL
LIN {X 0,Y 530.968,Z 417.343,A -85,B 0,C 180,E1 -4303.07,E2 -4303.07} C_VEL
LIN {X 0,Y 531.016,Z 417.334,A -85,B 0,C 180,E1 -4305.436,E2 -4305.436} C_VEL
LIN {X 0,Y 531.037,Z 417.34,A -85,B 0,C 180,E1 -4308.55,E2 -4308.55} C_VEL
LIN {X 0,Y 531.053,Z 417.329,A -85,B 0,C 180,E1 -4311.629,E2 -4311.629} C_VEL
LIN {X 0,Y 531.117,Z 417.33,A -85,B 0,C 180,E1 -4314.685,E2 -4314.685} C_VEL
LIN {X 0,Y 531.139,Z 417.318,A -85,B 0,C 180,E1 -4317.725,E2 -4317.725} C_VEL
LIN {X 0,Y 531.153,Z 417.325,A -85,B 0,C 180,E1 -4320.758,E2 -4320.758} C_VEL
LIN {X 0,Y 531.101,Z 417.327,A -85,B 0,C 180,E1 -4323.034,E2 -4323.034} C_VEL
LIN {X 0,Y 531.081,Z 417.327,A -85,B 0,C 180,E1 -4326.077,E2 -4326.077} C_VEL
LIN {X 0,Y 531.052,Z 417.334,A -85,B 0,C 180,E1 -4328.371,E2 -4328.371} C_VEL
LIN {X 0,Y 531.052,Z 417.329,A -85,B 0,C 180,E1 -4331.672,E2 -4331.672} C_VEL
LIN {X 0,Y 531.031,Z 417.337,A -85,B 0,C 180,E1 -4334.956,E2 -4334.956} C_VEL
LIN {X 0,Y 530.981,Z 417.338,A -85,B 0,C 180,E1 -4337.724,E2 -4337.724} C_VEL
LIN {X 0,Y 531.025,Z 417.334,A -85,B 0,C 180,E1 -4340.127,E2 -4340.127} C_VEL
LIN {X 0,Y 530.945,Z 417.35,A -85,B 0,C 180,E1 -4342.573,E2 -4342.573} C_VEL
LIN {X 0,Y 530.999,Z 417.34,A -85,B 0,C 180,E1 -4345.058,E2 -4345.058} C_VEL
LIN {X 0,Y 530.988,Z 417.337,A -85,B 0,C 180,E1 -4347.597,E2 -4347.597} C_VEL
LIN {X 0,Y 530.974,Z 417.348,A -85,B 0,C 180,E1 -4350.645,E2 -4350.645} C_VEL
LIN {X 0,Y 530.987,Z 417.337,A -85,B 0,C 180,E1 -4353.773,E2 -4353.773} C_VEL
LIN {X 0,Y 530.956,Z 417.348,A -85,B 0,C 180,E1 -4356.559,E2 -4356.559} C_VEL
LIN {X 0,Y 530.986,Z 417.338,A -85,B 0,C 180,E1 -4359.444,E2 -4359.444} C_VEL
LIN {X 0,Y 530.978,Z 417.344,A -85,B 0,C 180,E1 -4362.457,E2 -4362.457} C_VEL
LIN {X 0,Y 530.985,Z 417.338,A -85,B 0,C 180,E1 -4365.621,E2 -4365.621} C_VEL
LIN {X 0,Y 530.994,Z 417.343,A -85,B 0,C 180,E1 -4368.565,E2 -4368.565} C_VEL
LIN {X 0,Y 530.958,Z 417.341,A -85,B 0,C 180,E1 -4371.53,E2 -4371.53} C_VEL
LIN {X 0,Y 530.951,Z 417.346,A -85,B 0,C 180,E1 -4374.38,E2 -4374.38} C_VEL
LIN {X 0,Y 530.968,Z 417.344,A -85,B 0,C 180,E1 -4377.134,E2 -4377.134} C_VEL
LIN {X 0,Y 530.97,Z 417.34,A -85,B 0,C 180,E1 -4379.803,E2 -4379.803} C_VEL
LIN {X 0,Y 531.013,Z 417.342,A -85,B 0,C 180,E1 -4382.468,E2 -4382.468} C_VEL
LIN {X 0,Y 531.015,Z 417.531,A -85,B 0,C 180,E1 -4383.856,E2 -4383.856} C_VEL
LIN {X 0,Y 532.854,Z 427.292,A -85,B 0,C 180,E1 -4385.335,E2 -4385.335} C_VEL
LIN {X 0,Y 532.451,Z 443.701,A -85,B 0,C 180,E1 -4387.62,E2 -4387.62} C_VEL
LIN {X 0,Y 532.056,Z 464.864,A -85,B 0,C 180,E1 -4390.517,E2 -4390.517} C_VEL
LIN {X 0,Y 531.649,Z 486.845,A -85,B 0,C 180,E1 -4393.488,E2 -4393.488} C_VEL
LIN {X 0,Y 531.488,Z 498.692,A -85,B 0,C 180,E1 -4395.058,E2 -4395.058} C_VEL
LIN {X 0,Y 532.76,Z 508.639,A -85,B 0,C 180,E1 -4395.227,E2 -4395.227} C_VEL
LIN {X 0,Y 532.403,Z 606.953,A -85,B 0,C 180,E1 -4396.571,E2 -4396.571} C_VEL
LIN {X 0,Y 532.19,Z 620.494,A -85,B 0,C 180,E1 -4396.906,E2 -4396.906} C_VEL
LIN {X 0,Y 531.992,Z 632.815,A -85,B 0,C 180,E1 -4397.362,E2 -4397.362} C_VEL
LIN {X 0,Y 531.778,Z 644.745,A -85,B 0,C 180,E1 -4397.957,E2 -4397.957} C_VEL
LIN {X 0,Y 531.525,Z 656.949,A -85,B 0,C 180,E1 -4398.754,E2 -4398.754} C_VEL
LIN {X 0,Y 531.233,Z 667.486,A -85,B 0,C 180,E1 -4399.616,E2 -4399.616} C_VEL
LIN {X 0,Y 531.062,Z 676.096,A -85,B 0,C 180,E1 -4400.478,E2 -4400.478} C_VEL
LIN {X 0,Y 530.886,Z 683.962,A -85,B 0,C 180,E1 -4401.435,E2 -4401.435} C_VEL
LIN {X 0,Y 530.684,Z 691.622,A -85,B 0,C 180,E1 -4402.581,E2 -4402.581} C_VEL
LIN {X 0,Y 530.604,Z 698.68,A -85,B 0,C 180,E1 -4403.918,E2 -4403.918} C_VEL
LIN {X 0,Y 530.459,Z 703.374,A -85,B 0,C 180,E1 -4405.06,E2 -4405.06} C_VEL
LIN {X 0,Y 530.516,Z 706.958,A -85,B 0,C 180,E1 -4406.202,E2 -4406.202} C_VEL
LIN {X 0,Y 530.457,Z 708.807,A -85,B 0,C 180,E1 -4406.962,E2 -4406.962} C_VEL
LIN {X 0,Y 530.411,Z 710.193,A -85,B 0,C 180,E1 -4407.722,E2 -4407.722} C_VEL
LIN {X 0,Y 530.344,Z 711.785,A -85,B 0,C 180,E1 -4409.241,E2 -4409.241} C_VEL
LIN {X 0,Y 530.342,Z 712,A -85,B 0,C 180,E1 -4410,E2 -4410} C_VEL
LIN {X 0,Y 530.361,Z 711.183,A -85,B 0,C 180,E1 -4411.519,E2 -4411.519} C_VEL
LIN {X 0,Y 530.411,Z 710.195,A -85,B 0,C 180,E1 -4412.278,E2 -4412.278} C_VEL
LIN {X 0,Y 530.457,Z 708.809,A -85,B 0,C 180,E1 -4413.038,E2 -4413.038} C_VEL
LIN {X 0,Y 530.523,Z 705.894,A -85,B 0,C 180,E1 -4414.179,E2 -4414.179} C_VEL
LIN {X 0,Y 530.524,Z 701.947,A -85,B 0,C 180,E1 -4415.321,E2 -4415.321} C_VEL
LIN {X 0,Y 530.599,Z 696.261,A -85,B 0,C 180,E1 -4416.582,E2 -4416.582} C_VEL
LIN {X 0,Y 530.758,Z 689.233,A -85,B 0,C 180,E1 -4417.801,E2 -4417.801} C_VEL
LIN {X 0,Y 530.93,Z 680.989,A -85,B 0,C 180,E1 -4418.948,E2 -4418.948} C_VEL
LIN {X 0,Y 531.14,Z 672.483,A -85,B 0,C 180,E1 -4419.905,E2 -4419.905} C_VEL
LIN {X 0,Y 531.377,Z 661.878,A -85,B 0,C 180,E1 -4420.864,E2 -4420.864} C_VEL
LIN {X 0,Y 531.662,Z 651.002,A -85,B 0,C 180,E1 -4421.656,E2 -4421.656} C_VEL
LIN {X 0,Y 531.862,Z 639.862,A -85,B 0,C 180,E1 -4422.303,E2 -4422.303} C_VEL
LIN {X 0,Y 532.059,Z 627.99,A -85,B 0,C 180,E1 -4422.831,E2 -4422.831} C_VEL
LIN {X 0,Y 532.295,Z 614.308,A -85,B 0,C 180,E1 -4423.262,E2 -4423.262} C_VEL
LIN {X 0,Y 532.444,Z 602.147,A -85,B 0,C 180,E1 -4423.502,E2 -4423.502} C_VEL
LIN {X 0,Y 532.627,Z 506.875,A -85,B 0,C 180,E1 -4424.794,E2 -4424.794} C_VEL
LIN {X 0,Y 531.431,Z 498.057,A -85,B 0,C 180,E1 -4424.966,E2 -4424.966} C_VEL
LIN {X 0,Y 531.779,Z 475.958,A -85,B 0,C 180,E1 -4427.907,E2 -4427.907} C_VEL
LIN {X 0,Y 532.189,Z 453.81,A -85,B 0,C 180,E1 -4430.889,E2 -4430.889} C_VEL
LIN {X 0,Y 532.586,Z 431.5,A -85,B 0,C 180,E1 -4433.94,E2 -4433.94} C_VEL
LIN {X 0,Y 532.57,Z 425.195,A -85,B 0,C 180,E1 -4434.82,E2 -4434.82} C_VEL
LIN {X 0,Y 531.03,Z 417.338,A -85,B 0,C 180,E1 -4436.002,E2 -4436.002} C_VEL
LIN {X 0,Y 531.001,Z 417.341,A -85,B 0,C 180,E1 -4438.456,E2 -4438.456} C_VEL
LIN {X 0,Y 530.961,Z 417.352,A -85,B 0,C 180,E1 -4441.079,E2 -4441.079} C_VEL
LIN {X 0,Y 530.992,Z 417.342,A -85,B 0,C 180,E1 -4443.773,E2 -4443.773} C_VEL
LIN {X 0,Y 530.959,Z 417.348,A -85,B 0,C 180,E1 -4446.559,E2 -4446.559} C_VEL
LIN {X 0,Y 530.99,Z 417.341,A -85,B 0,C 180,E1 -4449.444,E2 -4449.444} C_VEL
LIN {X 0,Y 530.982,Z 417.344,A -85,B 0,C 180,E1 -4452.457,E2 -4452.457} C_VEL
LIN {X 0,Y 530.982,Z 417.339,A -85,B 0,C 180,E1 -4455.622,E2 -4455.622} C_VEL
LIN {X 0,Y 530.993,Z 417.346,A -85,B 0,C 180,E1 -4458.564,E2 -4458.564} C_VEL
LIN {X 0,Y 530.957,Z 417.342,A -85,B 0,C 180,E1 -4461.529,E2 -4461.529} C_VEL
LIN {X 0,Y 530.952,Z 417.349,A -85,B 0,C 180,E1 -4464.38,E2 -4464.38} C_VEL
LIN {X 0,Y 530.971,Z 417.341,A -85,B 0,C 180,E1 -4467.133,E2 -4467.133} C_VEL
LIN {X 0,Y 530.955,Z 417.344,A -85,B 0,C 180,E1 -4469.802,E2 -4469.802} C_VEL
LIN {X 0,Y 530.964,Z 417.349,A -85,B 0,C 180,E1 -4472.479,E2 -4472.479} C_VEL
LIN {X 0,Y 530.952,Z 417.344,A -85,B 0,C 180,E1 -4474.94,E2 -4474.94} C_VEL
LIN {X 0,Y 530.98,Z 417.344,A -85,B 0,C 180,E1 -4477.899,E2 -4477.899} C_VEL
LIN {X 0,Y 530.919,Z 417.349,A -85,B 0,C 180,E1 -4480.674,E2 -4480.674} C_VEL
LIN {X 0,Y 530.929,Z 417.346,A -85,B 0,C 180,E1 -4483.069,E2 -4483.069} C_VEL
LIN {X 0,Y 530.983,Z 417.341,A -85,B 0,C 180,E1 -4485.435,E2 -4485.435} C_VEL
LIN {X 0,Y 530.986,Z 417.341,A -85,B 0,C 180,E1 -4488.549,E2 -4488.549} C_VEL
LIN {X 0,Y 530.983,Z 417.345,A -85,B 0,C 180,E1 -4491.628,E2 -4491.628} C_VEL
LIN {X 0,Y 531.083,Z 417.329,A -85,B 0,C 180,E1 -4494.685,E2 -4494.685} C_VEL
LIN {X 0,Y 531.136,Z 417.329,A -85,B 0,C 180,E1 -4497.725,E2 -4497.725} C_VEL
LIN {X 0,Y 531.071,Z 417.491,A -85,B 0,C 180,E1 -4498.626,E2 -4498.626} C_VEL
LIN {X 0,Y 531.191,Z 421.697,A -85,B 0,C 180,E1 -4499.621,E2 -4499.621} C_VEL
LIN {X 0,Y 531.169,Z 423.829,A -85,B 0,C 180,E1 -4500.118,E2 -4500.118} C_VEL
LIN {X 0,Y 532.827,Z 432.954,A -85,B 0,C 180,E1 -4500.307,E2 -4500.307} C_VEL
LIN {X 0,Y 532.374,Z 529.6,A -85,B 0,C 180,E1 -4501.655,E2 -4501.655} C_VEL
LIN {X 0,Y 532.17,Z 541.634,A -85,B 0,C 180,E1 -4501.963,E2 -4501.963} C_VEL
LIN {X 0,Y 532.036,Z 552.648,A -85,B 0,C 180,E1 -4502.366,E2 -4502.366} C_VEL
LIN {X 0,Y 531.797,Z 564.377,A -85,B 0,C 180,E1 -4502.935,E2 -4502.935} C_VEL
LIN {X 0,Y 531.499,Z 576.316,A -85,B 0,C 180,E1 -4503.696,E2 -4503.696} C_VEL
LIN {X 0,Y 531.253,Z 585.803,A -85,B 0,C 180,E1 -4504.458,E2 -4504.458} C_VEL
LIN {X 0,Y 531.105,Z 594.571,A -85,B 0,C 180,E1 -4505.315,E2 -4505.315} C_VEL
LIN {X 0,Y 530.944,Z 601.197,A -85,B 0,C 180,E1 -4506.079,E2 -4506.079} C_VEL
LIN {X 0,Y 530.811,Z 608.166,A -85,B 0,C 180,E1 -4507.035,E2 -4507.035} C_VEL
LIN {X 0,Y 530.703,Z 613.986,A -85,B 0,C 180,E1 -4507.993,E2 -4507.993} C_VEL
LIN {X 0,Y 530.561,Z 619.7,A -85,B 0,C 180,E1 -4509.146,E2 -4509.146} C_VEL
LIN {X 0,Y 530.498,Z 624.208,A -85,B 0,C 180,E1 -4510.303,E2 -4510.303} C_VEL
LIN {X 0,Y 530.463,Z 627.632,A -85,B 0,C 180,E1 -4511.463,E2 -4511.463} C_VEL
LIN {X 0,Y 530.368,Z 630.638,A -85,B 0,C 180,E1 -4513.019,E2 -4513.019} C_VEL
LIN {X 0,Y 530.394,Z 631.526,A -85,B 0,C 180,E1 -4513.799,E2 -4513.799} C_VEL
LIN {X 0,Y 530.319,Z 631.97,A -85,B 0,C 180,E1 -4515.37,E2 -4515.37} C_VEL
LIN {X 0,Y 530.331,Z 631.648,A -85,B 0,C 180,E1 -4516.158,E2 -4516.158} C_VEL
LIN {X 0,Y 530.387,Z 629.505,A -85,B 0,C 180,E1 -4517.744,E2 -4517.744} C_VEL
LIN {X 0,Y 530.437,Z 626.761,A -85,B 0,C 180,E1 -4518.942,E2 -4518.942} C_VEL
LIN {X 0,Y 530.504,Z 622.9,A -85,B 0,C 180,E1 -4520.148,E2 -4520.148} C_VEL
LIN {X 0,Y 530.579,Z 617.796,A -85,B 0,C 180,E1 -4521.362,E2 -4521.362} C_VEL
LIN {X 0,Y 530.72,Z 611.208,A -85,B 0,C 180,E1 -4522.583,E2 -4522.583} C_VEL
LIN {X 0,Y 530.866,Z 604.485,A -85,B 0,C 180,E1 -4523.582,E2 -4523.582} C_VEL
LIN {X 0,Y 531.023,Z 597.689,A -85,B 0,C 180,E1 -4524.43,E2 -4524.43} C_VEL
LIN {X 0,Y 531.235,Z 588.682,A -85,B 0,C 180,E1 -4525.36,E2 -4525.36} C_VEL
LIN {X 0,Y 531.429,Z 580.247,A -85,B 0,C 180,E1 -4526.086,E2 -4526.086} C_VEL
LIN {X 0,Y 531.644,Z 571.577,A -85,B 0,C 180,E1 -4526.709,E2 -4526.709} C_VEL
LIN {X 0,Y 531.891,Z 560.89,A -85,B 0,C 180,E1 -4527.333,E2 -4527.333} C_VEL
LIN {X 0,Y 532.061,Z 550.86,A -85,B 0,C 180,E1 -4527.796,E2 -4527.796} C_VEL
LIN {X 0,Y 532.248,Z 539.161,A -85,B 0,C 180,E1 -4528.202,E2 -4528.202} C_VEL
LIN {X 0,Y 532.355,Z 526.954,A -85,B 0,C 180,E1 -4528.484,E2 -4528.484} C_VEL
LIN {X 0,Y 532.786,Z 439.196,A -85,B 0,C 180,E1 -4529.688,E2 -4529.688} C_VEL
LIN {X 0,Y 532.089,Z 437.057,A -85,B 0,C 180,E1 -4529.737,E2 -4529.737} C_VEL
LIN {X 0,Y 529.314,Z 434.324,A -85,B 0,C 180,E1 -4529.856,E2 -4529.856} C_VEL
LIN {X 0,Y 526.287,Z 431.646,A -85,B 0,C 180,E1 -4529.983,E2 -4529.983} C_VEL
LIN {X 0,Y 525.253,Z 429.53,A -85,B 0,C 180,E1 -4530.045,E2 -4530.045} C_VEL
LIN {X 0,Y 524.152,Z 423.85,A -85,B 0,C 180,E1 -4530.161,E2 -4530.161} C_VEL
LIN {X 0,Y 523.983,Z 418.217,A -85,B 0,C 180,E1 -4531.442,E2 -4531.442} C_VEL
LIN {X 0,Y 523.916,Z 418.227,A -85,B 0,C 180,E1 -4534.292,E2 -4534.292} C_VEL
LIN {X 0,Y 523.884,Z 418.223,A -85,B 0,C 180,E1 -4537.134,E2 -4537.134} C_VEL
LIN {X 0,Y 523.915,Z 418.224,A -85,B 0,C 180,E1 -4540.126,E2 -4540.126} C_VEL
LIN {X 0,Y 523.892,Z 418.222,A -85,B 0,C 180,E1 -4543.17,E2 -4543.17} C_VEL
LIN {X 0,Y 523.922,Z 418.219,A -85,B 0,C 180,E1 -4545.77,E2 -4545.77} C_VEL
LIN {X 0,Y 523.898,Z 418.223,A -85,B 0,C 180,E1 -4548.903,E2 -4548.903} C_VEL
LIN {X 0,Y 523.904,Z 418.222,A -85,B 0,C 180,E1 -4551.897,E2 -4551.897} C_VEL
LIN {X 0,Y 523.919,Z 418.22,A -85,B 0,C 180,E1 -4554.912,E2 -4554.912} C_VEL
LIN {X 0,Y 523.937,Z 418.216,A -85,B 0,C 180,E1 -4557.68,E2 -4557.68} C_VEL
LIN {X 0,Y 523.938,Z 418.221,A -85,B 0,C 180,E1 -4560.68,E2 -4560.68} C_VEL
LIN {X 0,Y 523.912,Z 418.219,A -85,B 0,C 180,E1 -4563.725,E2 -4563.725} C_VEL
LIN {X 0,Y 523.911,Z 418.226,A -85,B 0,C 180,E1 -4566.269,E2 -4566.269} C_VEL
LIN {X 0,Y 523.947,Z 418.219,A -85,B 0,C 180,E1 -4568.766,E2 -4568.766} C_VEL
LIN {X 0,Y 523.938,Z 418.216,A -85,B 0,C 180,E1 -4571.22,E2 -4571.22} C_VEL
LIN {X 0,Y 523.893,Z 418.221,A -85,B 0,C 180,E1 -4573.637,E2 -4573.637} C_VEL
LIN {X 0,Y 523.926,Z 418.22,A -85,B 0,C 180,E1 -4576.027,E2 -4576.027} C_VEL
LIN {X 0,Y 523.995,Z 418.209,A -85,B 0,C 180,E1 -4579.177,E2 -4579.177} C_VEL
LIN {X 0,Y 523.978,Z 418.217,A -85,B 0,C 180,E1 -4582.292,E2 -4582.292} C_VEL
LIN {X 0,Y 524.068,Z 418.207,A -85,B 0,C 180,E1 -4584.613,E2 -4584.613} C_VEL
LIN {X 0,Y 524.111,Z 418.194,A -85,B 0,C 180,E1 -4587.694,E2 -4587.694} C_VEL
LIN {X 0,Y 524.121,Z 418.198,A -85,B 0,C 180,E1 -4590.768,E2 -4590.768} C_VEL
LIN {X 0,Y 524.032,Z 418.205,A -85,B 0,C 180,E1 -4593.075,E2 -4593.075} C_VEL
LIN {X 0,Y 524.043,Z 418.207,A -85,B 0,C 180,E1 -4596.159,E2 -4596.159} C_VEL
LIN {X 0,Y 523.984,Z 418.21,A -85,B 0,C 180,E1 -4599.262,E2 -4599.262} C_VEL
LIN {X 0,Y 524.001,Z 418.208,A -85,B 0,C 180,E1 -4601.737,E2 -4601.737} C_VEL
LIN {X 0,Y 523.996,Z 418.21,A -85,B 0,C 180,E1 -4605.052,E2 -4605.052} C_VEL
LIN {X 0,Y 523.948,Z 418.216,A -85,B 0,C 180,E1 -4607.969,E2 -4607.969} C_VEL
LIN {X 0,Y 523.973,Z 418.219,A -85,B 0,C 180,E1 -4610.41,E2 -4610.41} C_VEL
LIN {X 0,Y 523.911,Z 418.223,A -85,B 0,C 180,E1 -4612.893,E2 -4612.893} C_VEL
LIN {X 0,Y 523.929,Z 418.217,A -85,B 0,C 180,E1 -4615.42,E2 -4615.42} C_VEL
LIN {X 0,Y 523.918,Z 418.22,A -85,B 0,C 180,E1 -4618.002,E2 -4618.002} C_VEL
LIN {X 0,Y 523.945,Z 418.219,A -85,B 0,C 180,E1 -4620.854,E2 -4620.854} C_VEL
LIN {X 0,Y 523.959,Z 418.213,A -85,B 0,C 180,E1 -4623.734,E2 -4623.734} C_VEL
LIN {X 0,Y 523.899,Z 418.227,A -85,B 0,C 180,E1 -4626.4,E2 -4626.4} C_VEL
LIN {X 0,Y 523.913,Z 418.221,A -85,B 0,C 180,E1 -4629.085,E2 -4629.085} C_VEL
LIN {X 0,Y 523.94,Z 418.218,A -85,B 0,C 180,E1 -4632.12,E2 -4632.12} C_VEL
LIN {X 0,Y 523.941,Z 418.216,A -85,B 0,C 180,E1 -4635.31,E2 -4635.31} C_VEL
LIN {X 0,Y 523.952,Z 418.221,A -85,B 0,C 180,E1 -4638.69,E2 -4638.69} C_VEL
LIN {X 0,Y 523.915,Z 418.221,A -85,B 0,C 180,E1 -4641.081,E2 -4641.081} C_VEL
LIN {X 0,Y 523.895,Z 418.221,A -85,B 0,C 180,E1 -4643.825,E2 -4643.825} C_VEL
LIN {X 0,Y 523.941,Z 418.224,A -85,B 0,C 180,E1 -4646.636,E2 -4646.636} C_VEL
LIN {X 0,Y 523.955,Z 418.214,A -85,B 0,C 180,E1 -4649.356,E2 -4649.356} C_VEL
LIN {X 0,Y 523.971,Z 418.216,A -85,B 0,C 180,E1 -4652.283,E2 -4652.283} C_VEL
LIN {X 0,Y 523.922,Z 418.218,A -85,B 0,C 180,E1 -4655.428,E2 -4655.428} C_VEL
LIN {X 0,Y 523.945,Z 418.222,A -85,B 0,C 180,E1 -4658.767,E2 -4658.767} C_VEL
LIN {X 0,Y 523.947,Z 418.216,A -85,B 0,C 180,E1 -4661.221,E2 -4661.221} C_VEL
LIN {X 0,Y 523.925,Z 418.217,A -85,B 0,C 180,E1 -4663.639,E2 -4663.639} C_VEL
LIN {X 0,Y 523.935,Z 418.217,A -85,B 0,C 180,E1 -4666.028,E2 -4666.028} C_VEL
LIN {X 0,Y 524.013,Z 418.212,A -85,B 0,C 180,E1 -4668.394,E2 -4668.394} C_VEL
LIN {X 0,Y 524,Z 418.208,A -85,B 0,C 180,E1 -4671.516,E2 -4671.516} C_VEL
LIN {X 0,Y 524.078,Z 418.207,A -85,B 0,C 180,E1 -4674.614,E2 -4674.614} C_VEL
LIN {X 0,Y 524.111,Z 418.194,A -85,B 0,C 180,E1 -4677.695,E2 -4677.695} C_VEL
LIN {X 0,Y 524.123,Z 418.2,A -85,B 0,C 180,E1 -4680.768,E2 -4680.768} C_VEL
LIN {X 0,Y 524.068,Z 418.203,A -85,B 0,C 180,E1 -4683.075,E2 -4683.075} C_VEL
LIN {X 0,Y 524.044,Z 418.205,A -85,B 0,C 180,E1 -4686.159,E2 -4686.159} C_VEL
LIN {X 0,Y 524,Z 418.214,A -85,B 0,C 180,E1 -4688.484,E2 -4688.484} C_VEL
LIN {X 0,Y 524.003,Z 418.207,A -85,B 0,C 180,E1 -4691.74,E2 -4691.74} C_VEL
LIN {X 0,Y 523.995,Z 418.212,A -85,B 0,C 180,E1 -4695.053,E2 -4695.053} C_VEL
LIN {X 0,Y 523.948,Z 418.215,A -85,B 0,C 180,E1 -4697.97,E2 -4697.97} C_VEL
LIN {X 0,Y 523.972,Z 418.216,A -85,B 0,C 180,E1 -4700.41,E2 -4700.41} C_VEL
LIN {X 0,Y 523.911,Z 418.225,A -85,B 0,C 180,E1 -4702.894,E2 -4702.894} C_VEL
LIN {X 0,Y 523.935,Z 418.216,A -85,B 0,C 180,E1 -4705.42,E2 -4705.42} C_VEL
LIN {X 0,Y 523.953,Z 418.214,A -85,B 0,C 180,E1 -4708,E2 -4708} C_VEL
LIN {X 0,Y 523.945,Z 418.222,A -85,B 0,C 180,E1 -4710.855,E2 -4710.855} C_VEL
LIN {X 0,Y 523.959,Z 418.213,A -85,B 0,C 180,E1 -4713.735,E2 -4713.735} C_VEL
LIN {X 0,Y 523.904,Z 418.224,A -85,B 0,C 180,E1 -4716.402,E2 -4716.402} C_VEL
LIN {X 0,Y 523.92,Z 418.222,A -85,B 0,C 180,E1 -4719.085,E2 -4719.085} C_VEL
LIN {X 0,Y 523.952,Z 418.215,A -85,B 0,C 180,E1 -4722.119,E2 -4722.119} C_VEL
LIN {X 0,Y 523.954,Z 418.215,A -85,B 0,C 180,E1 -4725.309,E2 -4725.309} C_VEL
LIN {X 0,Y 523.957,Z 418.222,A -85,B 0,C 180,E1 -4728.69,E2 -4728.69} C_VEL
LIN {X 0,Y 523.919,Z 418.222,A -85,B 0,C 180,E1 -4731.081,E2 -4731.081} C_VEL
LIN {X 0,Y 523.896,Z 418.221,A -85,B 0,C 180,E1 -4733.825,E2 -4733.825} C_VEL
LIN {X 0,Y 523.943,Z 418.223,A -85,B 0,C 180,E1 -4736.636,E2 -4736.636} C_VEL
LIN {X 0,Y 523.957,Z 418.216,A -85,B 0,C 180,E1 -4739.356,E2 -4739.356} C_VEL
LIN {X 0,Y 523.975,Z 418.217,A -85,B 0,C 180,E1 -4742.282,E2 -4742.282} C_VEL
LIN {X 0,Y 523.976,Z 418.322,A -85,B 0,C 180,E1 -4743.649,E2 -4743.649} C_VEL
LIN {X 0,Y 525.882,Z 427.697,A -85,B 0,C 180,E1 -4745.098,E2 -4745.098} C_VEL
LIN {X 0,Y 525.658,Z 440.907,A -85,B 0,C 180,E1 -4746.979,E2 -4746.979} C_VEL
LIN {X 0,Y 525.148,Z 461.512,A -85,B 0,C 180,E1 -4749.842,E2 -4749.842} C_VEL
LIN {X 0,Y 524.706,Z 483.509,A -85,B 0,C 180,E1 -4752.862,E2 -4752.862} C_VEL
LIN {X 0,Y 524.431,Z 498.229,A -85,B 0,C 180,E1 -4754.852,E2 -4754.852} C_VEL
LIN {X 0,Y 525.862,Z 508.983,A -85,B 0,C 180,E1 -4755.047,E2 -4755.047} C_VEL
LIN {X 0,Y 525.467,Z 605.732,A -85,B 0,C 180,E1 -4756.39,E2 -4756.39} C_VEL
LIN {X 0,Y 525.285,Z 618.832,A -85,B 0,C 180,E1 -4756.706,E2 -4756.706} C_VEL
LIN {X 0,Y 525.012,Z 632.01,A -85,B 0,C 180,E1 -4757.191,E2 -4757.191} C_VEL
LIN {X 0,Y 524.782,Z 644.326,A -85,B 0,C 180,E1 -4757.812,E2 -4757.812} C_VEL
LIN {X 0,Y 524.515,Z 656.27,A -85,B 0,C 180,E1 -4758.602,E2 -4758.602} C_VEL
LIN {X 0,Y 524.2,Z 666.838,A -85,B 0,C 180,E1 -4759.475,E2 -4759.475} C_VEL
LIN {X 0,Y 524.005,Z 675.486,A -85,B 0,C 180,E1 -4760.349,E2 -4760.349} C_VEL
LIN {X 0,Y 523.808,Z 683.462,A -85,B 0,C 180,E1 -4761.319,E2 -4761.319} C_VEL
LIN {X 0,Y 523.616,Z 691.25,A -85,B 0,C 180,E1 -4762.481,E2 -4762.481} C_VEL
LIN {X 0,Y 523.495,Z 698.425,A -85,B 0,C 180,E1 -4763.835,E2 -4763.835} C_VEL
LIN {X 0,Y 523.383,Z 703.196,A -85,B 0,C 180,E1 -4764.993,E2 -4764.993} C_VEL
LIN {X 0,Y 523.443,Z 706.851,A -85,B 0,C 180,E1 -4766.151,E2 -4766.151} C_VEL
LIN {X 0,Y 523.367,Z 708.728,A -85,B 0,C 180,E1 -4766.921,E2 -4766.921} C_VEL
LIN {X 0,Y 523.335,Z 710.136,A -85,B 0,C 180,E1 -4767.691,E2 -4767.691} C_VEL
LIN {X 0,Y 523.25,Z 711.747,A -85,B 0,C 180,E1 -4769.231,E2 -4769.231} C_VEL
LIN {X 0,Y 523.246,Z 711.964,A -85,B 0,C 180,E1 -4770,E2 -4770} C_VEL
LIN {X 0,Y 523.274,Z 711.138,A -85,B 0,C 180,E1 -4771.54,E2 -4771.54} C_VEL
LIN {X 0,Y 523.335,Z 710.138,A -85,B 0,C 180,E1 -4772.309,E2 -4772.309} C_VEL
LIN {X 0,Y 523.368,Z 708.73,A -85,B 0,C 180,E1 -4773.079,E2 -4773.079} C_VEL
LIN {X 0,Y 523.425,Z 705.763,A -85,B 0,C 180,E1 -4774.235,E2 -4774.235} C_VEL
LIN {X 0,Y 523.464,Z 701.741,A -85,B 0,C 180,E1 -4775.393,E2 -4775.393} C_VEL
LIN {X 0,Y 523.524,Z 696.416,A -85,B 0,C 180,E1 -4776.581,E2 -4776.581} C_VEL
LIN {X 0,Y 523.665,Z 690.033,A -85,B 0,C 180,E1 -4777.713,E2 -4777.713} C_VEL
LIN {X 0,Y 523.845,Z 681.892,A -85,B 0,C 180,E1 -4778.876,E2 -4778.876} C_VEL
LIN {X 0,Y 524.055,Z 673.59,A -85,B 0,C 180,E1 -4779.846,E2 -4779.846} C_VEL
LIN {X 0,Y 524.307,Z 663.455,A -85,B 0,C 180,E1 -4780.817,E2 -4780.817} C_VEL
LIN {X 0,Y 524.601,Z 652.009,A -85,B 0,C 180,E1 -4781.69,E2 -4781.69} C_VEL
LIN {X 0,Y 524.814,Z 640.748,A -85,B 0,C 180,E1 -4782.373,E2 -4782.373} C_VEL
LIN {X 0,Y 525.082,Z 628.243,A -85,B 0,C 180,E1 -4782.956,E2 -4782.956} C_VEL
LIN {X 0,Y 525.323,Z 614.929,A -85,B 0,C 180,E1 -4783.392,E2 -4783.392} C_VEL
LIN {X 0,Y 525.503,Z 602.073,A -85,B 0,C 180,E1 -4783.659,E2 -4783.659} C_VEL
LIN {X 0,Y 525.748,Z 507.602,A -85,B 0,C 180,E1 -4784.966,E2 -4784.966} C_VEL
LIN {X 0,Y 524.373,Z 497.355,A -85,B 0,C 180,E1 -4785.178,E2 -4785.178} C_VEL
LIN {X 0,Y 524.77,Z 475.548,A -85,B 0,C 180,E1 -4788.122,E2 -4788.122} C_VEL
LIN {X 0,Y 525.236,Z 453.176,A -85,B 0,C 180,E1 -4791.179,E2 -4791.179} C_VEL
LIN {X 0,Y 525.689,Z 430.92,A -85,B 0,C 180,E1 -4794.274,E2 -4794.274} C_VEL
LIN {X 0,Y 525.575,Z 426.313,A -85,B 0,C 180,E1 -4794.931,E2 -4794.931} C_VEL
LIN {X 0,Y 523.973,Z 418.217,A -85,B 0,C 180,E1 -4796.19,E2 -4796.19} C_VEL
LIN {X 0,Y 523.943,Z 418.223,A -85,B 0,C 180,E1 -4798.875,E2 -4798.875} C_VEL
LIN {X 0,Y 523.925,Z 418.225,A -85,B 0,C 180,E1 -4801.544,E2 -4801.544} C_VEL
LIN {X 0,Y 523.941,Z 418.221,A -85,B 0,C 180,E1 -4804.29,E2 -4804.29} C_VEL
LIN {X 0,Y 523.911,Z 418.227,A -85,B 0,C 180,E1 -4807.132,E2 -4807.132} C_VEL
LIN {X 0,Y 523.942,Z 418.218,A -85,B 0,C 180,E1 -4810.13,E2 -4810.13} C_VEL
LIN {X 0,Y 523.939,Z 418.222,A -85,B 0,C 180,E1 -4812.459,E2 -4812.459} C_VEL
LIN {X 0,Y 523.949,Z 418.216,A -85,B 0,C 180,E1 -4815.31,E2 -4815.31} C_VEL
LIN {X 0,Y 523.957,Z 418.222,A -85,B 0,C 180,E1 -4818.69,E2 -4818.69} C_VEL
LIN {X 0,Y 523.919,Z 418.221,A -85,B 0,C 180,E1 -4821.081,E2 -4821.081} C_VEL
LIN {X 0,Y 523.898,Z 418.222,A -85,B 0,C 180,E1 -4823.825,E2 -4823.825} C_VEL
LIN {X 0,Y 523.945,Z 418.221,A -85,B 0,C 180,E1 -4826.636,E2 -4826.636} C_VEL
LIN {X 0,Y 523.948,Z 418.215,A -85,B 0,C 180,E1 -4829.355,E2 -4829.355} C_VEL
LIN {X 0,Y 523.921,Z 418.226,A -85,B 0,C 180,E1 -4832.294,E2 -4832.294} C_VEL
LIN {X 0,Y 523.906,Z 418.221,A -85,B 0,C 180,E1 -4835.427,E2 -4835.427} C_VEL
LIN {X 0,Y 523.94,Z 418.222,A -85,B 0,C 180,E1 -4837.939,E2 -4837.939} C_VEL
LIN {X 0,Y 523.904,Z 418.226,A -85,B 0,C 180,E1 -4840.405,E2 -4840.405} C_VEL
LIN {X 0,Y 523.897,Z 418.223,A -85,B 0,C 180,E1 -4842.835,E2 -4842.835} C_VEL
LIN {X 0,Y 523.927,Z 418.219,A -85,B 0,C 180,E1 -4845.234,E2 -4845.234} C_VEL
LIN {X 0,Y 523.961,Z 418.218,A -85,B 0,C 180,E1 -4848.393,E2 -4848.393} C_VEL
LIN {X 0,Y 523.947,Z 418.221,A -85,B 0,C 180,E1 -4851.515,E2 -4851.515} C_VEL
LIN {X 0,Y 524.029,Z 418.208,A -85,B 0,C 180,E1 -4854.613,E2 -4854.613} C_VEL
LIN {X 0,Y 524.046,Z 418.212,A -85,B 0,C 180,E1 -4858.079,E2 -4858.079} C_VEL
